LIN {X 0,Y 185.451,Z 180.384,A -85,B 0,C 180,E1 -22369.893,E2 -22369.893} C_VEL
LIN {X 0,Y 185.61,Z 180.474,A -85,B 0,C 180,E1 -22373.267,E2 -22373.267} C_VEL
LIN {X 0,Y 186.703,Z 185.931,A -85,B 0,C 180,E1 -22376.028,E2 -22376.028} C_VEL
LIN {X 0,Y 194.99,Z 213.07,A -85,B 0,C 180,E1 -22378.383,E2 -22378.383} C_VEL
LIN {X 0,Y 197.604,Z 239.191,A -85,B 0,C 180,E1 -22379.998,E2 -22379.998} C_VEL
LIN {X 0,Y 195.443,Z 280.522,A -85,B 0,C 180,E1 -22381.986,E2 -22381.986} C_VEL
LIN {X 0,Y 194.473,Z 286.295,A -85,B 0,C 180,E1 -22382.216,E2 -22382.216} C_VEL
LIN {X 0,Y 191.045,Z 295.55,A -85,B 0,C 180,E1 -22382.527,E2 -22382.527} C_VEL
LIN {X 0,Y 187.492,Z 304.682,A -85,B 0,C 180,E1 -22383.032,E2 -22383.032} C_VEL
LIN {X 0,Y 186.3,Z 310.262,A -85,B 0,C 180,E1 -22383.531,E2 -22383.531} C_VEL
LIN {X 0,Y 184.548,Z 324.129,A -85,B 0,C 180,E1 -22385.237,E2 -22385.237} C_VEL
LIN {X 0,Y 182.934,Z 335.61,A -85,B 0,C 180,E1 -22387.111,E2 -22387.111} C_VEL
LIN {X 0,Y 181.066,Z 347.271,A -85,B 0,C 180,E1 -22389.556,E2 -22389.556} C_VEL
LIN {X 0,Y 179.457,Z 357.77,A -85,B 0,C 180,E1 -22392.334,E2 -22392.334} C_VEL
LIN {X 0,Y 178.167,Z 366.277,A -85,B 0,C 180,E1 -22395.145,E2 -22395.145} C_VEL
LIN {X 0,Y 177.112,Z 374.602,A -85,B 0,C 180,E1 -22398.558,E2 -22398.558} C_VEL
LIN {X 0,Y 176.53,Z 381.268,A -85,B 0,C 180,E1 -22401.992,E2 -22401.992} C_VEL
LIN {X 0,Y 176.349,Z 386.5,A -85,B 0,C 180,E1 -22405.43,E2 -22405.43} C_VEL
LIN {X 0,Y 176.332,Z 390.477,A -85,B 0,C 180,E1 -22408.86,E2 -22408.86} C_VEL
LIN {X 0,Y 176.266,Z 393.307,A -85,B 0,C 180,E1 -22412.287,E2 -22412.287} C_VEL
LIN {X 0,Y 176.184,Z 395.515,A -85,B 0,C 180,E1 -22416.875,E2 -22416.875} C_VEL
LIN {X 0,Y 177.166,Z 396.208,A -85,B 0,C 180,E1 -22421.442,E2 -22421.442} C_VEL
LIN {X 0,Y 179.11,Z 395.354,A -85,B 0,C 180,E1 -22425.944,E2 -22425.944} C_VEL
LIN {X 0,Y 182.326,Z 392.981,A -85,B 0,C 180,E1 -22430.301,E2 -22430.301} C_VEL
LIN {X 0,Y 185.623,Z 390.146,A -85,B 0,C 180,E1 -22433.427,E2 -22433.427} C_VEL
LIN {X 0,Y 190.628,Z 384.946,A -85,B 0,C 180,E1 -22437.444,E2 -22437.444} C_VEL
LIN {X 0,Y 195.03,Z 379.819,A -85,B 0,C 180,E1 -22440.3,E2 -22440.3} C_VEL
LIN {X 0,Y 200.108,Z 373.441,A -85,B 0,C 180,E1 -22442.984,E2 -22442.984} C_VEL
LIN {X 0,Y 206.708,Z 364.199,A -85,B 0,C 180,E1 -22445.911,E2 -22445.911} C_VEL
LIN {X 0,Y 211.819,Z 356.151,A -85,B 0,C 180,E1 -22447.868,E2 -22447.868} C_VEL
LIN {X 0,Y 217.199,Z 346.506,A -85,B 0,C 180,E1 -22449.723,E2 -22449.723} C_VEL
LIN {X 0,Y 222.849,Z 334.573,A -85,B 0,C 180,E1 -22451.476,E2 -22451.476} C_VEL
LIN {X 0,Y 227.689,Z 322.728,A -85,B 0,C 180,E1 -22452.773,E2 -22452.773} C_VEL
LIN {X 0,Y 231.851,Z 310.219,A -85,B 0,C 180,E1 -22453.751,E2 -22453.751} C_VEL
LIN {X 0,Y 235.139,Z 297.091,A -85,B 0,C 180,E1 -22454.54,E2 -22454.54} C_VEL
LIN {X 0,Y 237.675,Z 281.593,A -85,B 0,C 180,E1 -22455.21,E2 -22455.21} C_VEL
LIN {X 0,Y 240.135,Z 263.541,A -85,B 0,C 180,E1 -22455.927,E2 -22455.927} C_VEL
LIN {X 0,Y 238.425,Z 258.199,A -85,B 0,C 180,E1 -22457.785,E2 -22457.785} C_VEL
LIN {X 0,Y 236.912,Z 254.032,A -85,B 0,C 180,E1 -22459.595,E2 -22459.595} C_VEL
LIN {X 0,Y 235.86,Z 251.223,A -85,B 0,C 180,E1 -22461.183,E2 -22461.183} C_VEL
LIN {X 0,Y 234.74,Z 248.234,A -85,B 0,C 180,E1 -22463.217,E2 -22463.217} C_VEL
LIN {X 0,Y 233.654,Z 245.558,A -85,B 0,C 180,E1 -22466.277,E2 -22466.277} C_VEL
LIN {X 0,Y 233.421,Z 244.65,A -85,B 0,C 180,E1 -22468.158,E2 -22468.158} C_VEL
LIN {X 0,Y 233.575,Z 244.599,A -85,B 0,C 180,E1 -22471.222,E2 -22471.222} C_VEL
LIN {X 0,Y 234.571,Z 246.09,A -85,B 0,C 180,E1 -22474.401,E2 -22474.401} C_VEL
LIN {X 0,Y 235.287,Z 247.149,A -85,B 0,C 180,E1 -22475.846,E2 -22475.846} C_VEL
LIN {X 0,Y 237.14,Z 250.744,A -85,B 0,C 180,E1 -22478.579,E2 -22478.579} C_VEL
LIN {X 0,Y 239.474,Z 255.65,A -85,B 0,C 180,E1 -22481.167,E2 -22481.167} C_VEL
LIN {X 0,Y 240.686,Z 258.623,A -85,B 0,C 180,E1 -22482.374,E2 -22482.374} C_VEL
LIN {X 0,Y 236.176,Z 289.327,A -85,B 0,C 180,E1 -22483.584,E2 -22483.584} C_VEL
LIN {X 0,Y 233.164,Z 302.706,A -85,B 0,C 180,E1 -22484.372,E2 -22484.372} C_VEL
LIN {X 0,Y 229.525,Z 314.723,A -85,B 0,C 180,E1 -22485.368,E2 -22485.368} C_VEL
LIN {X 0,Y 225.29,Z 326.032,A -85,B 0,C 180,E1 -22486.61,E2 -22486.61} C_VEL
LIN {X 0,Y 220.162,Z 337.516,A -85,B 0,C 180,E1 -22488.259,E2 -22488.259} C_VEL
LIN {X 0,Y 214.619,Z 347.927,A -85,B 0,C 180,E1 -22490.19,E2 -22490.19} C_VEL
LIN {X 0,Y 209.255,Z 356.656,A -85,B 0,C 180,E1 -22492.28,E2 -22492.28} C_VEL
LIN {X 0,Y 204.148,Z 363.965,A -85,B 0,C 180,E1 -22494.518,E2 -22494.518} C_VEL
LIN {X 0,Y 198.214,Z 371.419,A -85,B 0,C 180,E1 -22497.46,E2 -22497.46} C_VEL
LIN {X 0,Y 192.399,Z 377.919,A -85,B 0,C 180,E1 -22501.047,E2 -22501.047} C_VEL
LIN {X 0,Y 188.037,Z 382.07,A -85,B 0,C 180,E1 -22504.287,E2 -22504.287} C_VEL
LIN {X 0,Y 184.361,Z 385.041,A -85,B 0,C 180,E1 -22507.62,E2 -22507.62} C_VEL
LIN {X 0,Y 181.286,Z 386.968,A -85,B 0,C 180,E1 -22511.177,E2 -22511.177} C_VEL
LIN {X 0,Y 179.696,Z 387.622,A -85,B 0,C 180,E1 -22513.572,E2 -22513.572} C_VEL
LIN {X 0,Y 177.448,Z 387.679,A -85,B 0,C 180,E1 -22518.089,E2 -22518.089} C_VEL
LIN {X 0,Y 176.483,Z 386.859,A -85,B 0,C 180,E1 -22521.003,E2 -22521.003} C_VEL
LIN {X 0,Y 175.945,Z 385.646,A -85,B 0,C 180,E1 -22523.544,E2 -22523.544} C_VEL
LIN {X 0,Y 175.632,Z 383.889,A -85,B 0,C 180,E1 -22526.116,E2 -22526.116} C_VEL
LIN {X 0,Y 175.734,Z 380.218,A -85,B 0,C 180,E1 -22529.994,E2 -22529.994} C_VEL
LIN {X 0,Y 176.17,Z 375.043,A -85,B 0,C 180,E1 -22533.953,E2 -22533.953} C_VEL
LIN {X 0,Y 176.776,Z 369.274,A -85,B 0,C 180,E1 -22537.33,E2 -22537.33} C_VEL
LIN {X 0,Y 177.741,Z 361.636,A -85,B 0,C 180,E1 -22540.862,E2 -22540.862} C_VEL
LIN {X 0,Y 179.054,Z 352.651,A -85,B 0,C 180,E1 -22544.164,E2 -22544.164} C_VEL
LIN {X 0,Y 180.522,Z 343.259,A -85,B 0,C 180,E1 -22546.947,E2 -22546.947} C_VEL
LIN {X 0,Y 182.287,Z 331.812,A -85,B 0,C 180,E1 -22549.638,E2 -22549.638} C_VEL
LIN {X 0,Y 183.88,Z 321.431,A -85,B 0,C 180,E1 -22551.585,E2 -22551.585} C_VEL
LIN {X 0,Y 185.496,Z 309.195,A -85,B 0,C 180,E1 -22553.394,E2 -22553.394} C_VEL
LIN {X 0,Y 186.884,Z 295.677,A -85,B 0,C 180,E1 -22554.88,E2 -22554.88} C_VEL
LIN {X 0,Y 187.935,Z 282.298,A -85,B 0,C 180,E1 -22555.898,E2 -22555.898} C_VEL
LIN {X 0,Y 191.478,Z 219.149,A -85,B 0,C 180,E1 -22559.077,E2 -22559.077} C_VEL
LIN {X 0,Y 184.988,Z 198.355,A -85,B 0,C 180,E1 -22560.871,E2 -22560.871} C_VEL
LIN {X 0,Y 178.472,Z 181.316,A -85,B 0,C 180,E1 -22562.595,E2 -22562.595} C_VEL
LIN {X 0,Y 178.468,Z 181.254,A -85,B 0,C 180,E1 -22566.807,E2 -22566.807} C_VEL
LIN {X 0,Y 178.61,Z 181.237,A -85,B 0,C 180,E1 -22571.65,E2 -22571.65} C_VEL
LIN {X 0,Y 178.631,Z 181.236,A -85,B 0,C 180,E1 -22576.344,E2 -22576.344} C_VEL
LIN {X 0,Y 178.909,Z 181.198,A -85,B 0,C 180,E1 -22580.958,E2 -22580.958} C_VEL
LIN {X 0,Y 179.127,Z 181.172,A -85,B 0,C 180,E1 -22587.75,E2 -22587.75} C_VEL
LIN {X 0,Y 179.348,Z 181.141,A -85,B 0,C 180,E1 -22589.998,E2 -22589.998} C_VEL
LIN {X 0,Y 178.836,Z 181.207,A -85,B 0,C 180,E1 -22594.506,E2 -22594.506} C_VEL
LIN {X 0,Y 178.905,Z 181.194,A -85,B 0,C 180,E1 -22599.039,E2 -22599.039} C_VEL
LIN {X 0,Y 178.628,Z 181.234,A -85,B 0,C 180,E1 -22603.652,E2 -22603.652} C_VEL
LIN {X 0,Y 178.555,Z 181.242,A -85,B 0,C 180,E1 -22609.15,E2 -22609.15} C_VEL
LIN {X 0,Y 178.465,Z 181.251,A -85,B 0,C 180,E1 -22615.074,E2 -22615.074} C_VEL
LIN {X 0,Y 178.459,Z 181.255,A -85,B 0,C 180,E1 -22620.792,E2 -22620.792} C_VEL
LIN {X 0,Y 178.481,Z 181.247,A -85,B 0,C 180,E1 -22624.216,E2 -22624.216} C_VEL
LIN {X 0,Y 178.385,Z 181.265,A -85,B 0,C 180,E1 -22629.075,E2 -22629.075} C_VEL
LIN {X 0,Y 178.39,Z 181.257,A -85,B 0,C 180,E1 -22632.044,E2 -22632.044} C_VEL
LIN {X 0,Y 178.388,Z 181.265,A -85,B 0,C 180,E1 -22635.163,E2 -22635.163} C_VEL
LIN {X 0,Y 178.394,Z 181.263,A -85,B 0,C 180,E1 -22638.46,E2 -22638.46} C_VEL
LIN {X 0,Y 178.415,Z 181.259,A -85,B 0,C 180,E1 -22643.78,E2 -22643.78} C_VEL
LIN {X 0,Y 178.479,Z 181.253,A -85,B 0,C 180,E1 -22646.544,E2 -22646.544} C_VEL
LIN {X 0,Y 178.435,Z 181.257,A -85,B 0,C 180,E1 -22651.793,E2 -22651.793} C_VEL
LIN {X 0,Y 178.5,Z 181.248,A -85,B 0,C 180,E1 -22654.895,E2 -22654.895} C_VEL
LIN {X 0,Y 178.6,Z 181.237,A -85,B 0,C 180,E1 -22661.65,E2 -22661.65} C_VEL
LIN {X 0,Y 178.62,Z 181.233,A -85,B 0,C 180,E1 -22666.344,E2 -22666.344} C_VEL
LIN {X 0,Y 178.899,Z 181.199,A -85,B 0,C 180,E1 -22670.959,E2 -22670.959} C_VEL
LIN {X 0,Y 179.117,Z 181.174,A -85,B 0,C 180,E1 -22677.751,E2 -22677.751} C_VEL
LIN {X 0,Y 179.338,Z 181.145,A -85,B 0,C 180,E1 -22679.999,E2 -22679.999} C_VEL
LIN {X 0,Y 178.826,Z 181.208,A -85,B 0,C 180,E1 -22684.508,E2 -22684.508} C_VEL
LIN {X 0,Y 178.896,Z 181.198,A -85,B 0,C 180,E1 -22689.041,E2 -22689.041} C_VEL
LIN {X 0,Y 178.619,Z 181.236,A -85,B 0,C 180,E1 -22693.655,E2 -22693.655} C_VEL
LIN {X 0,Y 178.548,Z 181.24,A -85,B 0,C 180,E1 -22699.152,E2 -22699.152} C_VEL
LIN {X 0,Y 178.459,Z 181.255,A -85,B 0,C 180,E1 -22705.077,E2 -22705.077} C_VEL
LIN {X 0,Y 178.454,Z 181.255,A -85,B 0,C 180,E1 -22710.795,E2 -22710.795} C_VEL
LIN {X 0,Y 178.476,Z 181.25,A -85,B 0,C 180,E1 -22714.219,E2 -22714.219} C_VEL
LIN {X 0,Y 178.381,Z 181.265,A -85,B 0,C 180,E1 -22719.078,E2 -22719.078} C_VEL
LIN {X 0,Y 178.387,Z 181.261,A -85,B 0,C 180,E1 -22722.048,E2 -22722.048} C_VEL
LIN {X 0,Y 178.386,Z 181.267,A -85,B 0,C 180,E1 -22725.166,E2 -22725.166} C_VEL
LIN {X 0,Y 178.392,Z 181.264,A -85,B 0,C 180,E1 -22728.463,E2 -22728.463} C_VEL
LIN {X 0,Y 178.548,Z 181.257,A -85,B 0,C 180,E1 -22732.828,E2 -22732.828} C_VEL
LIN {X 0,Y 179.513,Z 185.981,A -85,B 0,C 180,E1 -22735.227,E2 -22735.227} C_VEL
LIN {X 0,Y 188.36,Z 214.966,A -85,B 0,C 180,E1 -22737.833,E2 -22737.833} C_VEL
LIN {X 0,Y 190.739,Z 240.435,A -85,B 0,C 180,E1 -22739.459,E2 -22739.459} C_VEL
LIN {X 0,Y 187.702,Z 294.949,A -85,B 0,C 180,E1 -22742.247,E2 -22742.247} C_VEL
LIN {X 0,Y 186.444,Z 309.054,A -85,B 0,C 180,E1 -22743.411,E2 -22743.411} C_VEL
LIN {X 0,Y 186.3,Z 310.262,A -85,B 0,C 180,E1 -22743.531,E2 -22743.531} C_VEL
LIN {X 0,Y 184.978,Z 315.739,A -85,B 0,C 180,E1 -22744.087,E2 -22744.087} C_VEL
LIN {X 0,Y 181.018,Z 324.289,A -85,B 0,C 180,E1 -22745.068,E2 -22745.068} C_VEL
LIN {X 0,Y 176.974,Z 332.538,A -85,B 0,C 180,E1 -22746.295,E2 -22746.295} C_VEL
LIN {X 0,Y 175.539,Z 337.528,A -85,B 0,C 180,E1 -22747.221,E2 -22747.221} C_VEL
LIN {X 0,Y 173.85,Z 348.124,A -85,B 0,C 180,E1 -22749.596,E2 -22749.596} C_VEL
LIN {X 0,Y 172.373,Z 357.468,A -85,B 0,C 180,E1 -22752.197,E2 -22752.197} C_VEL
LIN {X 0,Y 171.057,Z 365.993,A -85,B 0,C 180,E1 -22755.123,E2 -22755.123} C_VEL
LIN {X 0,Y 170.019,Z 374.338,A -85,B 0,C 180,E1 -22758.679,E2 -22758.679} C_VEL
LIN {X 0,Y 169.512,Z 379.97,A -85,B 0,C 180,E1 -22761.658,E2 -22761.658} C_VEL
LIN {X 0,Y 169.295,Z 385.409,A -85,B 0,C 180,E1 -22765.24,E2 -22765.24} C_VEL
LIN {X 0,Y 169.279,Z 389.572,A -85,B 0,C 180,E1 -22768.813,E2 -22768.813} C_VEL
LIN {X 0,Y 169.198,Z 392.583,A -85,B 0,C 180,E1 -22772.383,E2 -22772.383} C_VEL
LIN {X 0,Y 169.039,Z 394.032,A -85,B 0,C 180,E1 -22774.772,E2 -22774.772} C_VEL
LIN {X 0,Y 169.129,Z 395.073,A -85,B 0,C 180,E1 -22777.163,E2 -22777.163} C_VEL
LIN {X 0,Y 170.184,Z 395.952,A -85,B 0,C 180,E1 -22781.918,E2 -22781.918} C_VEL
LIN {X 0,Y 172.265,Z 395.359,A -85,B 0,C 180,E1 -22786.596,E2 -22786.596} C_VEL
LIN {X 0,Y 173.807,Z 394.504,A -85,B 0,C 180,E1 -22788.876,E2 -22788.876} C_VEL
LIN {X 0,Y 177.963,Z 391.591,A -85,B 0,C 180,E1 -22793.263,E2 -22793.263} C_VEL
LIN {X 0,Y 182.975,Z 387.134,A -85,B 0,C 180,E1 -22797.448,E2 -22797.448} C_VEL
LIN {X 0,Y 187.391,Z 382.606,A -85,B 0,C 180,E1 -22800.419,E2 -22800.419} C_VEL
LIN {X 0,Y 193.364,Z 375.929,A -85,B 0,C 180,E1 -22803.663,E2 -22803.663} C_VEL
LIN {X 0,Y 200.141,Z 367.459,A -85,B 0,C 180,E1 -22806.654,E2 -22806.654} C_VEL
LIN {X 0,Y 206.443,Z 358.412,A -85,B 0,C 180,E1 -22809.037,E2 -22809.037} C_VEL
LIN {X 0,Y 213.139,Z 347.295,A -85,B 0,C 180,E1 -22811.262,E2 -22811.262} C_VEL
LIN {X 0,Y 218.411,Z 337.106,A -85,B 0,C 180,E1 -22812.826,E2 -22812.826} C_VEL
LIN {X 0,Y 223.4,Z 325.833,A -85,B 0,C 180,E1 -22814.112,E2 -22814.112} C_VEL
LIN {X 0,Y 227.963,Z 313.355,A -85,B 0,C 180,E1 -22815.162,E2 -22815.162} C_VEL
LIN {X 0,Y 231.687,Z 299.909,A -85,B 0,C 180,E1 -22816.014,E2 -22816.014} C_VEL
LIN {X 0,Y 234.426,Z 286.088,A -85,B 0,C 180,E1 -22816.635,E2 -22816.635} C_VEL
LIN {X 0,Y 237.134,Z 267.255,A -85,B 0,C 180,E1 -22817.403,E2 -22817.403} C_VEL
LIN {X 0,Y 235.477,Z 261.867,A -85,B 0,C 180,E1 -22819.489,E2 -22819.489} C_VEL
LIN {X 0,Y 234.173,Z 257.979,A -85,B 0,C 180,E1 -22821.561,E2 -22821.561} C_VEL
LIN {X 0,Y 233.184,Z 255.014,A -85,B 0,C 180,E1 -22823.577,E2 -22823.577} C_VEL
LIN {X 0,Y 232.217,Z 252.288,A -85,B 0,C 180,E1 -22826.767,E2 -22826.767} C_VEL
LIN {X 0,Y 231.999,Z 251.475,A -85,B 0,C 180,E1 -22829.004,E2 -22829.004} C_VEL
LIN {X 0,Y 232.373,Z 251.836,A -85,B 0,C 180,E1 -22832.071,E2 -22832.071} C_VEL
LIN {X 0,Y 233.663,Z 253.817,A -85,B 0,C 180,E1 -22835.382,E2 -22835.382} C_VEL
LIN {X 0,Y 235.34,Z 257.377,A -85,B 0,C 180,E1 -22838.103,E2 -22838.103} C_VEL
LIN {X 0,Y 237.32,Z 261.821,A -85,B 0,C 180,E1 -22840.504,E2 -22840.504} C_VEL
LIN {X 0,Y 237.707,Z 262.858,A -85,B 0,C 180,E1 -22840.939,E2 -22840.939} C_VEL
LIN {X 0,Y 233.439,Z 289.877,A -85,B 0,C 180,E1 -22841.995,E2 -22841.995} C_VEL
LIN {X 0,Y 230.262,Z 303.162,A -85,B 0,C 180,E1 -22842.772,E2 -22842.772} C_VEL
LIN {X 0,Y 226.388,Z 315.434,A -85,B 0,C 180,E1 -22843.776,E2 -22843.776} C_VEL
LIN {X 0,Y 221.725,Z 327.318,A -85,B 0,C 180,E1 -22845.076,E2 -22845.076} C_VEL
LIN {X 0,Y 216.772,Z 337.743,A -85,B 0,C 180,E1 -22846.571,E2 -22846.571} C_VEL
LIN {X 0,Y 210.976,Z 348.019,A -85,B 0,C 180,E1 -22848.471,E2 -22848.471} C_VEL
LIN {X 0,Y 205.104,Z 357.104,A -85,B 0,C 180,E1 -22850.633,E2 -22850.633} C_VEL
LIN {X 0,Y 198.669,Z 365.689,A -85,B 0,C 180,E1 -22853.334,E2 -22853.334} C_VEL
LIN {X 0,Y 193.399,Z 371.78,A -85,B 0,C 180,E1 -22855.833,E2 -22855.833} C_VEL
LIN {X 0,Y 188.003,Z 377.408,A -85,B 0,C 180,E1 -22858.929,E2 -22858.929} C_VEL
LIN {X 0,Y 182.893,Z 382,A -85,B 0,C 180,E1 -22862.394,E2 -22862.394} C_VEL
LIN {X 0,Y 180.269,Z 384.023,A -85,B 0,C 180,E1 -22864.473,E2 -22864.473} C_VEL
LIN {X 0,Y 177.186,Z 386.081,A -85,B 0,C 180,E1 -22867.413,E2 -22867.413} C_VEL
LIN {X 0,Y 173.706,Z 387.76,A -85,B 0,C 180,E1 -22871.672,E2 -22871.672} C_VEL
LIN {X 0,Y 172.112,Z 388.066,A -85,B 0,C 180,E1 -22874.183,E2 -22874.183} C_VEL
LIN {X 0,Y 170.235,Z 387.622,A -85,B 0,C 180,E1 -22878.274,E2 -22878.274} C_VEL
LIN {X 0,Y 169.152,Z 386.232,A -85,B 0,C 180,E1 -22881.959,E2 -22881.959} C_VEL
LIN {X 0,Y 168.56,Z 383.621,A -85,B 0,C 180,E1 -22885.964,E2 -22885.964} C_VEL
LIN {X 0,Y 168.652,Z 379.764,A -85,B 0,C 180,E1 -22890.005,E2 -22890.005} C_VEL
LIN {X 0,Y 169.046,Z 374.941,A -85,B 0,C 180,E1 -22893.745,E2 -22893.745} C_VEL
LIN {X 0,Y 169.727,Z 368.633,A -85,B 0,C 180,E1 -22897.522,E2 -22897.522} C_VEL
LIN {X 0,Y 170.732,Z 360.824,A -85,B 0,C 180,E1 -22901.196,E2 -22901.196} C_VEL
LIN {X 0,Y 172.003,Z 352.301,A -85,B 0,C 180,E1 -22904.406,E2 -22904.406} C_VEL
LIN {X 0,Y 173.493,Z 342.963,A -85,B 0,C 180,E1 -22907.243,E2 -22907.243} C_VEL
LIN {X 0,Y 175.382,Z 331.03,A -85,B 0,C 180,E1 -22910.119,E2 -22910.119} C_VEL
LIN {X 0,Y 177.023,Z 320.439,A -85,B 0,C 180,E1 -22912.139,E2 -22912.139} C_VEL
LIN {X 0,Y 178.669,Z 307.992,A -85,B 0,C 180,E1 -22913.985,E2 -22913.985} C_VEL
LIN {X 0,Y 179.945,Z 295.833,A -85,B 0,C 180,E1 -22915.35,E2 -22915.35} C_VEL
LIN {X 0,Y 181.03,Z 282.582,A -85,B 0,C 180,E1 -22916.395,E2 -22916.395} C_VEL
LIN {X 0,Y 184.658,Z 220.397,A -85,B 0,C 180,E1 -22919.648,E2 -22919.648} C_VEL
LIN {X 0,Y 178.39,Z 200.423,A -85,B 0,C 180,E1 -22921.463,E2 -22921.463} C_VEL
LIN {X 0,Y 171.445,Z 182.365,A -85,B 0,C 180,E1 -22923.382,E2 -22923.382} C_VEL
LIN {X 0,Y 171.394,Z 182.136,A -85,B 0,C 180,E1 -22923.559,E2 -22923.559} C_VEL
LIN {X 0,Y 171.42,Z 182.134,A -85,B 0,C 180,E1 -22928.345,E2 -22928.345} C_VEL
LIN {X 0,Y 171.513,Z 182.121,A -85,B 0,C 180,E1 -22930.862,E2 -22930.862} C_VEL
LIN {X 0,Y 171.546,Z 182.117,A -85,B 0,C 180,E1 -22935.768,E2 -22935.768} C_VEL
LIN {X 0,Y 171.848,Z 182.078,A -85,B 0,C 180,E1 -22940.583,E2 -22940.583} C_VEL
LIN {X 0,Y 171.787,Z 182.085,A -85,B 0,C 180,E1 -22945.305,E2 -22945.305} C_VEL
LIN {X 0,Y 172.313,Z 182.017,A -85,B 0,C 180,E1 -22949.998,E2 -22949.998} C_VEL
LIN {X 0,Y 171.785,Z 182.085,A -85,B 0,C 180,E1 -22954.691,E2 -22954.691} C_VEL
LIN {X 0,Y 171.844,Z 182.075,A -85,B 0,C 180,E1 -22959.413,E2 -22959.413} C_VEL
LIN {X 0,Y 171.543,Z 182.115,A -85,B 0,C 180,E1 -22964.228,E2 -22964.228} C_VEL
LIN {X 0,Y 171.48,Z 182.125,A -85,B 0,C 180,E1 -22969.497,E2 -22969.497} C_VEL
LIN {X 0,Y 171.403,Z 182.131,A -85,B 0,C 180,E1 -22975.567,E2 -22975.567} C_VEL
LIN {X 0,Y 171.416,Z 182.132,A -85,B 0,C 180,E1 -22980.57,E2 -22980.57} C_VEL
LIN {X 0,Y 171.39,Z 182.133,A -85,B 0,C 180,E1 -22985.033,E2 -22985.033} C_VEL
LIN {X 0,Y 171.341,Z 182.143,A -85,B 0,C 180,E1 -22988.799,E2 -22988.799} C_VEL
LIN {X 0,Y 171.315,Z 182.143,A -85,B 0,C 180,E1 -22994.216,E2 -22994.216} C_VEL
LIN {X 0,Y 171.326,Z 182.141,A -85,B 0,C 180,E1 -22998.978,E2 -22998.978} C_VEL
LIN {X 0,Y 171.356,Z 182.137,A -85,B 0,C 180,E1 -23002.032,E2 -23002.032} C_VEL
LIN {X 0,Y 171.393,Z 182.135,A -85,B 0,C 180,E1 -23005.091,E2 -23005.091} C_VEL
LIN {X 0,Y 171.403,Z 182.133,A -85,B 0,C 180,E1 -23010.525,E2 -23010.525} C_VEL
LIN {X 0,Y 171.421,Z 182.129,A -85,B 0,C 180,E1 -23015.795,E2 -23015.795} C_VEL
LIN {X 0,Y 171.501,Z 182.122,A -85,B 0,C 180,E1 -23020.862,E2 -23020.862} C_VEL
LIN {X 0,Y 171.536,Z 182.112,A -85,B 0,C 180,E1 -23025.769,E2 -23025.769} C_VEL
LIN {X 0,Y 171.837,Z 182.079,A -85,B 0,C 180,E1 -23030.584,E2 -23030.584} C_VEL
LIN {X 0,Y 171.777,Z 182.084,A -85,B 0,C 180,E1 -23035.306,E2 -23035.306} C_VEL
LIN {X 0,Y 172.303,Z 182.021,A -85,B 0,C 180,E1 -23039.999,E2 -23039.999} C_VEL
LIN {X 0,Y 171.775,Z 182.086,A -85,B 0,C 180,E1 -23044.693,E2 -23044.693} C_VEL
LIN {X 0,Y 171.835,Z 182.079,A -85,B 0,C 180,E1 -23049.415,E2 -23049.415} C_VEL
LIN {X 0,Y 171.535,Z 182.117,A -85,B 0,C 180,E1 -23054.23,E2 -23054.23} C_VEL
LIN {X 0,Y 171.472,Z 182.122,A -85,B 0,C 180,E1 -23059.499,E2 -23059.499} C_VEL
LIN {X 0,Y 171.396,Z 182.133,A -85,B 0,C 180,E1 -23065.57,E2 -23065.57} C_VEL
LIN {X 0,Y 171.411,Z 182.132,A -85,B 0,C 180,E1 -23070.573,E2 -23070.573} C_VEL
LIN {X 0,Y 171.386,Z 182.133,A -85,B 0,C 180,E1 -23075.036,E2 -23075.036} C_VEL
LIN {X 0,Y 171.337,Z 182.141,A -85,B 0,C 180,E1 -23078.802,E2 -23078.802} C_VEL
LIN {X 0,Y 171.313,Z 182.145,A -85,B 0,C 180,E1 -23084.22,E2 -23084.22} C_VEL
LIN {X 0,Y 171.331,Z 182.145,A -85,B 0,C 180,E1 -23088.983,E2 -23088.983} C_VEL
LIN {X 0,Y 171.508,Z 182.251,A -85,B 0,C 180,E1 -23092.497,E2 -23092.497} C_VEL
LIN {X 0,Y 172.164,Z 185.558,A -85,B 0,C 180,E1 -23094.317,E2 -23094.317} C_VEL
LIN {X 0,Y 181.585,Z 216.234,A -85,B 0,C 180,E1 -23097.236,E2 -23097.236} C_VEL
LIN {X 0,Y 183.928,Z 240.636,A -85,B 0,C 180,E1 -23098.865,E2 -23098.865} C_VEL
LIN {X 0,Y 180.825,Z 294.391,A -85,B 0,C 180,E1 -23101.729,E2 -23101.729} C_VEL
LIN {X 0,Y 179.534,Z 308.569,A -85,B 0,C 180,E1 -23102.933,E2 -23102.933} C_VEL
LIN {X 0,Y 177.851,Z 321.835,A -85,B 0,C 180,E1 -23104.551,E2 -23104.551} C_VEL
LIN {X 0,Y 176.19,Z 333.749,A -85,B 0,C 180,E1 -23106.494,E2 -23106.494} C_VEL
LIN {X 0,Y 175.539,Z 337.528,A -85,B 0,C 180,E1 -23107.221,E2 -23107.221} C_VEL
LIN {X 0,Y 174.103,Z 342.397,A -85,B 0,C 180,E1 -23108.217,E2 -23108.217} C_VEL
LIN {X 0,Y 170.033,Z 349.848,A -85,B 0,C 180,E1 -23109.934,E2 -23109.934} C_VEL
LIN {X 0,Y 166.024,Z 356.816,A -85,B 0,C 180,E1 -23111.934,E2 -23111.934} C_VEL
LIN {X 0,Y 164.712,Z 360.93,A -85,B 0,C 180,E1 -23113.341,E2 -23113.341} C_VEL
LIN {X 0,Y 163.358,Z 370.011,A -85,B 0,C 180,E1 -23116.948,E2 -23116.948} C_VEL
LIN {X 0,Y 162.615,Z 377.488,A -85,B 0,C 180,E1 -23120.675,E2 -23120.675} C_VEL
LIN {X 0,Y 162.298,Z 382.505,A -85,B 0,C 180,E1 -23123.787,E2 -23123.787} C_VEL
LIN {X 0,Y 162.244,Z 387.316,A -85,B 0,C 180,E1 -23127.519,E2 -23127.519} C_VEL
LIN {X 0,Y 162.24,Z 389.86,A -85,B 0,C 180,E1 -23130.002,E2 -23130.002} C_VEL
LIN {X 0,Y 161.983,Z 392.671,A -85,B 0,C 180,E1 -23133.71,E2 -23133.71} C_VEL
LIN {X 0,Y 162.098,Z 394.534,A -85,B 0,C 180,E1 -23137.476,E2 -23137.476} C_VEL
LIN {X 0,Y 163.225,Z 395.693,A -85,B 0,C 180,E1 -23142.434,E2 -23142.434} C_VEL
LIN {X 0,Y 165.447,Z 395.307,A -85,B 0,C 180,E1 -23147.301,E2 -23147.301} C_VEL
LIN {X 0,Y 169.103,Z 393.479,A -85,B 0,C 180,E1 -23151.967,E2 -23151.967} C_VEL
LIN {X 0,Y 171.491,Z 391.995,A -85,B 0,C 180,E1 -23154.196,E2 -23154.196} C_VEL
LIN {X 0,Y 176.728,Z 387.778,A -85,B 0,C 180,E1 -23158.505,E2 -23158.505} C_VEL
LIN {X 0,Y 181.368,Z 383.558,A -85,B 0,C 180,E1 -23161.543,E2 -23161.543} C_VEL
LIN {X 0,Y 187.591,Z 377.251,A -85,B 0,C 180,E1 -23164.845,E2 -23164.845} C_VEL
LIN {X 0,Y 193.59,Z 370.456,A -85,B 0,C 180,E1 -23167.453,E2 -23167.453} C_VEL
LIN {X 0,Y 200.024,Z 362.238,A -85,B 0,C 180,E1 -23169.886,E2 -23169.886} C_VEL
LIN {X 0,Y 206.894,Z 352.111,A -85,B 0,C 180,E1 -23172.138,E2 -23172.138} C_VEL
LIN {X 0,Y 212.875,Z 341.811,A -85,B 0,C 180,E1 -23173.894,E2 -23173.894} C_VEL
LIN {X 0,Y 218.568,Z 330.325,A -85,B 0,C 180,E1 -23175.353,E2 -23175.353} C_VEL
LIN {X 0,Y 223.207,Z 319.278,A -85,B 0,C 180,E1 -23176.403,E2 -23176.403} C_VEL
LIN {X 0,Y 227.608,Z 306.194,A -85,B 0,C 180,E1 -23177.332,E2 -23177.332} C_VEL
LIN {X 0,Y 231.046,Z 292.161,A -85,B 0,C 180,E1 -23178.041,E2 -23178.041} C_VEL
LIN {X 0,Y 234.386,Z 271.211,A -85,B 0,C 180,E1 -23178.864,E2 -23178.864} C_VEL
LIN {X 0,Y 233.018,Z 266.387,A -85,B 0,C 180,E1 -23181.018,E2 -23181.018} C_VEL
LIN {X 0,Y 231.649,Z 261.786,A -85,B 0,C 180,E1 -23183.924,E2 -23183.924} C_VEL
LIN {X 0,Y 230.821,Z 259.194,A -85,B 0,C 180,E1 -23186.995,E2 -23186.995} C_VEL
LIN {X 0,Y 230.659,Z 258.477,A -85,B 0,C 180,E1 -23188.804,E2 -23188.804} C_VEL
LIN {X 0,Y 230.988,Z 258.777,A -85,B 0,C 180,E1 -23191.93,E2 -23191.93} C_VEL
LIN {X 0,Y 232.152,Z 260.749,A -85,B 0,C 180,E1 -23195.14,E2 -23195.14} C_VEL
LIN {X 0,Y 233.627,Z 264.097,A -85,B 0,C 180,E1 -23197.711,E2 -23197.711} C_VEL
LIN {X 0,Y 234.856,Z 267.276,A -85,B 0,C 180,E1 -23199.458,E2 -23199.458} C_VEL
LIN {X 0,Y 231.009,Z 290.555,A -85,B 0,C 180,E1 -23200.357,E2 -23200.357} C_VEL
LIN {X 0,Y 227.791,Z 303.503,A -85,B 0,C 180,E1 -23201.098,E2 -23201.098} C_VEL
LIN {X 0,Y 223.556,Z 316.172,A -85,B 0,C 180,E1 -23202.122,E2 -23202.122} C_VEL
LIN {X 0,Y 218.614,Z 328.041,A -85,B 0,C 180,E1 -23203.423,E2 -23203.423} C_VEL
LIN {X 0,Y 213.191,Z 338.777,A -85,B 0,C 180,E1 -23204.956,E2 -23204.956} C_VEL
LIN {X 0,Y 207.341,Z 348.666,A -85,B 0,C 180,E1 -23206.774,E2 -23206.774} C_VEL
LIN {X 0,Y 201.095,Z 357.757,A -85,B 0,C 180,E1 -23208.955,E2 -23208.955} C_VEL
LIN {X 0,Y 194.206,Z 366.295,A -85,B 0,C 180,E1 -23211.677,E2 -23211.677} C_VEL
LIN {X 0,Y 187.74,Z 373.271,A -85,B 0,C 180,E1 -23214.63,E2 -23214.63} C_VEL
LIN {X 0,Y 182.081,Z 378.629,A -85,B 0,C 180,E1 -23217.788,E2 -23217.788} C_VEL
LIN {X 0,Y 177.166,Z 382.574,A -85,B 0,C 180,E1 -23220.999,E2 -23220.999} C_VEL
LIN {X 0,Y 172.579,Z 385.649,A -85,B 0,C 180,E1 -23224.672,E2 -23224.672} C_VEL
LIN {X 0,Y 170.012,Z 387.004,A -85,B 0,C 180,E1 -23227.185,E2 -23227.185} C_VEL
LIN {X 0,Y 167.902,Z 387.863,A -85,B 0,C 180,E1 -23229.639,E2 -23229.639} C_VEL
LIN {X 0,Y 165.743,Z 388.299,A -85,B 0,C 180,E1 -23232.761,E2 -23232.761} C_VEL
LIN {X 0,Y 163.354,Z 387.746,A -85,B 0,C 180,E1 -23237.528,E2 -23237.528} C_VEL
LIN {X 0,Y 162.446,Z 386.779,A -85,B 0,C 180,E1 -23240.25,E2 -23240.25} C_VEL
LIN {X 0,Y 161.665,Z 384.617,A -85,B 0,C 180,E1 -23244.083,E2 -23244.083} C_VEL
LIN {X 0,Y 161.505,Z 380.779,A -85,B 0,C 180,E1 -23248.6,E2 -23248.6} C_VEL
LIN {X 0,Y 161.849,Z 375.697,A -85,B 0,C 180,E1 -23252.875,E2 -23252.875} C_VEL
LIN {X 0,Y 162.44,Z 370.09,A -85,B 0,C 180,E1 -23256.51,E2 -23256.51} C_VEL
LIN {X 0,Y 163.321,Z 362.959,A -85,B 0,C 180,E1 -23260.203,E2 -23260.203} C_VEL
LIN {X 0,Y 164.667,Z 353.792,A -85,B 0,C 180,E1 -23263.948,E2 -23263.948} C_VEL
LIN {X 0,Y 166.096,Z 345.142,A -85,B 0,C 180,E1 -23266.803,E2 -23266.803} C_VEL
LIN {X 0,Y 167.894,Z 333.796,A -85,B 0,C 180,E1 -23269.814,E2 -23269.814} C_VEL
LIN {X 0,Y 169.833,Z 321.676,A -85,B 0,C 180,E1 -23272.32,E2 -23272.32} C_VEL
LIN {X 0,Y 171.547,Z 309.484,A -85,B 0,C 180,E1 -23274.262,E2 -23274.262} C_VEL
LIN {X 0,Y 172.949,Z 296.709,A -85,B 0,C 180,E1 -23275.783,E2 -23275.783} C_VEL
LIN {X 0,Y 174.033,Z 283.689,A -85,B 0,C 180,E1 -23276.885,E2 -23276.885} C_VEL
LIN {X 0,Y 177.806,Z 221.62,A -85,B 0,C 180,E1 -23280.267,E2 -23280.267} C_VEL
LIN {X 0,Y 171.897,Z 202.689,A -85,B 0,C 180,E1 -23282.069,E2 -23282.069} C_VEL
LIN {X 0,Y 164.414,Z 183.222,A -85,B 0,C 180,E1 -23284.216,E2 -23284.216} C_VEL
LIN {X 0,Y 164.361,Z 183.013,A -85,B 0,C 180,E1 -23284.683,E2 -23284.683} C_VEL
LIN {X 0,Y 164.421,Z 183.006,A -85,B 0,C 180,E1 -23290.116,E2 -23290.116} C_VEL
LIN {X 0,Y 164.476,Z 182.997,A -85,B 0,C 180,E1 -23295.143,E2 -23295.143} C_VEL
LIN {X 0,Y 164.769,Z 182.961,A -85,B 0,C 180,E1 -23300.174,E2 -23300.174} C_VEL
LIN {X 0,Y 164.824,Z 182.953,A -85,B 0,C 180,E1 -23302.649,E2 -23302.649} C_VEL
LIN {X 0,Y 165.277,Z 182.893,A -85,B 0,C 180,E1 -23309.998,E2 -23309.998} C_VEL
LIN {X 0,Y 164.821,Z 182.952,A -85,B 0,C 180,E1 -23317.347,E2 -23317.347} C_VEL
LIN {X 0,Y 164.703,Z 182.967,A -85,B 0,C 180,E1 -23321.055,E2 -23321.055} C_VEL
LIN {X 0,Y 164.429,Z 182.999,A -85,B 0,C 180,E1 -23327.407,E2 -23327.407} C_VEL
LIN {X 0,Y 164.42,Z 183.003,A -85,B 0,C 180,E1 -23329.994,E2 -23329.994} C_VEL
LIN {X 0,Y 164.338,Z 183.01,A -85,B 0,C 180,E1 -23336.092,E2 -23336.092} C_VEL
LIN {X 0,Y 164.352,Z 183.012,A -85,B 0,C 180,E1 -23341.212,E2 -23341.212} C_VEL
LIN {X 0,Y 164.278,Z 183.021,A -85,B 0,C 180,E1 -23346.791,E2 -23346.791} C_VEL
LIN {X 0,Y 164.283,Z 183.018,A -85,B 0,C 180,E1 -23349.916,E2 -23349.916} C_VEL
LIN {X 0,Y 164.277,Z 183.02,A -85,B 0,C 180,E1 -23353.34,E2 -23353.34} C_VEL
LIN {X 0,Y 164.257,Z 183.026,A -85,B 0,C 180,E1 -23356.796,E2 -23356.796} C_VEL
LIN {X 0,Y 164.285,Z 183.016,A -85,B 0,C 180,E1 -23360.353,E2 -23360.353} C_VEL
LIN {X 0,Y 164.321,Z 183.016,A -85,B 0,C 180,E1 -23364.349,E2 -23364.349} C_VEL
LIN {X 0,Y 164.362,Z 183.007,A -85,B 0,C 180,E1 -23369.128,E2 -23369.128} C_VEL
LIN {X 0,Y 164.381,Z 183.008,A -85,B 0,C 180,E1 -23374.687,E2 -23374.687} C_VEL
LIN {X 0,Y 164.411,Z 183.005,A -85,B 0,C 180,E1 -23380.116,E2 -23380.116} C_VEL
LIN {X 0,Y 164.465,Z 182.992,A -85,B 0,C 180,E1 -23385.143,E2 -23385.143} C_VEL
LIN {X 0,Y 164.759,Z 182.963,A -85,B 0,C 180,E1 -23390.175,E2 -23390.175} C_VEL
LIN {X 0,Y 164.814,Z 182.951,A -85,B 0,C 180,E1 -23392.65,E2 -23392.65} C_VEL
LIN {X 0,Y 165.267,Z 182.897,A -85,B 0,C 180,E1 -23399.999,E2 -23399.999} C_VEL
LIN {X 0,Y 164.811,Z 182.955,A -85,B 0,C 180,E1 -23407.349,E2 -23407.349} C_VEL
LIN {X 0,Y 164.694,Z 182.964,A -85,B 0,C 180,E1 -23411.057,E2 -23411.057} C_VEL
LIN {X 0,Y 164.421,Z 183.002,A -85,B 0,C 180,E1 -23417.409,E2 -23417.409} C_VEL
LIN {X 0,Y 164.412,Z 183.002,A -85,B 0,C 180,E1 -23419.996,E2 -23419.996} C_VEL
LIN {X 0,Y 164.332,Z 183.011,A -85,B 0,C 180,E1 -23426.095,E2 -23426.095} C_VEL
LIN {X 0,Y 164.351,Z 183.014,A -85,B 0,C 180,E1 -23431.218,E2 -23431.218} C_VEL
LIN {X 0,Y 164.274,Z 183.016,A -85,B 0,C 180,E1 -23436.794,E2 -23436.794} C_VEL
LIN {X 0,Y 164.28,Z 183.021,A -85,B 0,C 180,E1 -23439.919,E2 -23439.919} C_VEL
LIN {X 0,Y 164.274,Z 183.022,A -85,B 0,C 180,E1 -23443.343,E2 -23443.343} C_VEL
LIN {X 0,Y 164.255,Z 183.026,A -85,B 0,C 180,E1 -23446.799,E2 -23446.799} C_VEL
LIN {X 0,Y 164.409,Z 183.118,A -85,B 0,C 180,E1 -23452.088,E2 -23452.088} C_VEL
LIN {X 0,Y 164.897,Z 185.339,A -85,B 0,C 180,E1 -23453.37,E2 -23453.37} C_VEL
LIN {X 0,Y 172.786,Z 210.72,A -85,B 0,C 180,E1 -23455.957,E2 -23455.957} C_VEL
LIN {X 0,Y 175.078,Z 218.871,A -85,B 0,C 180,E1 -23456.712,E2 -23456.712} C_VEL
LIN {X 0,Y 177.083,Z 241.327,A -85,B 0,C 180,E1 -23458.263,E2 -23458.263} C_VEL
LIN {X 0,Y 173.898,Z 294.773,A -85,B 0,C 180,E1 -23461.24,E2 -23461.24} C_VEL
LIN {X 0,Y 172.642,Z 308.09,A -85,B 0,C 180,E1 -23462.418,E2 -23462.418} C_VEL
LIN {X 0,Y 170.905,Z 321.426,A -85,B 0,C 180,E1 -23464.095,E2 -23464.095} C_VEL
LIN {X 0,Y 169.216,Z 333.343,A -85,B 0,C 180,E1 -23466.106,E2 -23466.106} C_VEL
LIN {X 0,Y 167.42,Z 344.27,A -85,B 0,C 180,E1 -23468.452,E2 -23468.452} C_VEL
LIN {X 0,Y 165.64,Z 355.164,A -85,B 0,C 180,E1 -23471.447,E2 -23471.447} C_VEL
LIN {X 0,Y 164.712,Z 360.93,A -85,B 0,C 180,E1 -23473.341,E2 -23473.341} C_VEL
LIN {X 0,Y 163.455,Z 364.908,A -85,B 0,C 180,E1 -23474.823,E2 -23474.823} C_VEL
LIN {X 0,Y 159.752,Z 370.665,A -85,B 0,C 180,E1 -23477.357,E2 -23477.357} C_VEL
LIN {X 0,Y 156.267,Z 375.908,A -85,B 0,C 180,E1 -23480.16,E2 -23480.16} C_VEL
LIN {X 0,Y 155.383,Z 378.936,A -85,B 0,C 180,E1 -23482.011,E2 -23482.011} C_VEL
LIN {X 0,Y 155.199,Z 385.152,A -85,B 0,C 180,E1 -23486.444,E2 -23486.444} C_VEL
LIN {X 0,Y 155.193,Z 388.906,A -85,B 0,C 180,E1 -23490.002,E2 -23490.002} C_VEL
LIN {X 0,Y 154.952,Z 391.83,A -85,B 0,C 180,E1 -23493.778,E2 -23493.778} C_VEL
LIN {X 0,Y 155.083,Z 393.967,A -85,B 0,C 180,E1 -23497.816,E2 -23497.816} C_VEL
LIN {X 0,Y 156.288,Z 395.35,A -85,B 0,C 180,E1 -23502.996,E2 -23502.996} C_VEL
LIN {X 0,Y 158.659,Z 395.263,A -85,B 0,C 180,E1 -23508.066,E2 -23508.066} C_VEL
LIN {X 0,Y 162.557,Z 393.665,A -85,B 0,C 180,E1 -23512.901,E2 -23512.901} C_VEL
LIN {X 0,Y 167.668,Z 390.59,A -85,B 0,C 180,E1 -23517.459,E2 -23517.459} C_VEL
LIN {X 0,Y 172.861,Z 386.67,A -85,B 0,C 180,E1 -23521.171,E2 -23521.171} C_VEL
LIN {X 0,Y 179.016,Z 381.269,A -85,B 0,C 180,E1 -23524.701,E2 -23524.701} C_VEL
LIN {X 0,Y 186.001,Z 374.411,A -85,B 0,C 180,E1 -23527.881,E2 -23527.881} C_VEL
LIN {X 0,Y 192.518,Z 367.123,A -85,B 0,C 180,E1 -23530.391,E2 -23530.391} C_VEL
LIN {X 0,Y 199.448,Z 358.216,A -85,B 0,C 180,E1 -23532.714,E2 -23532.714} C_VEL
LIN {X 0,Y 206.804,Z 347.243,A -85,B 0,C 180,E1 -23534.845,E2 -23534.845} C_VEL
LIN {X 0,Y 212.528,Z 337.237,A -85,B 0,C 180,E1 -23536.336,E2 -23536.336} C_VEL
LIN {X 0,Y 217.9,Z 326.23,A -85,B 0,C 180,E1 -23537.546,E2 -23537.546} C_VEL
LIN {X 0,Y 223.06,Z 313.286,A -85,B 0,C 180,E1 -23538.574,E2 -23538.574} C_VEL
LIN {X 0,Y 226.639,Z 301.74,A -85,B 0,C 180,E1 -23539.299,E2 -23539.299} C_VEL
LIN {X 0,Y 229.842,Z 287.641,A -85,B 0,C 180,E1 -23539.927,E2 -23539.927} C_VEL
LIN {X 0,Y 231.807,Z 275.295,A -85,B 0,C 180,E1 -23540.455,E2 -23540.455} C_VEL
LIN {X 0,Y 230.714,Z 271.173,A -85,B 0,C 180,E1 -23542.549,E2 -23542.549} C_VEL
LIN {X 0,Y 230.028,Z 268.366,A -85,B 0,C 180,E1 -23544.514,E2 -23544.514} C_VEL
LIN {X 0,Y 229.438,Z 266.144,A -85,B 0,C 180,E1 -23547.144,E2 -23547.144} C_VEL
LIN {X 0,Y 229.278,Z 265.441,A -85,B 0,C 180,E1 -23549.126,E2 -23549.126} C_VEL
LIN {X 0,Y 229.658,Z 265.837,A -85,B 0,C 180,E1 -23552.092,E2 -23552.092} C_VEL
LIN {X 0,Y 230.652,Z 267.656,A -85,B 0,C 180,E1 -23554.896,E2 -23554.896} C_VEL
LIN {X 0,Y 231.946,Z 270.918,A -85,B 0,C 180,E1 -23557.364,E2 -23557.364} C_VEL
LIN {X 0,Y 232.276,Z 272.102,A -85,B 0,C 180,E1 -23557.952,E2 -23557.952} C_VEL
LIN {X 0,Y 228.916,Z 290.993,A -85,B 0,C 180,E1 -23558.671,E2 -23558.671} C_VEL
LIN {X 0,Y 225.439,Z 304.176,A -85,B 0,C 180,E1 -23559.413,E2 -23559.413} C_VEL
LIN {X 0,Y 220.777,Z 317.471,A -85,B 0,C 180,E1 -23560.474,E2 -23560.474} C_VEL
LIN {X 0,Y 215.406,Z 329.628,A -85,B 0,C 180,E1 -23561.808,E2 -23561.808} C_VEL
LIN {X 0,Y 210.061,Z 339.591,A -85,B 0,C 180,E1 -23563.228,E2 -23563.228} C_VEL
LIN {X 0,Y 203.63,Z 349.764,A -85,B 0,C 180,E1 -23565.107,E2 -23565.107} C_VEL
LIN {X 0,Y 197.47,Z 358.237,A -85,B 0,C 180,E1 -23567.148,E2 -23567.148} C_VEL
LIN {X 0,Y 191.277,Z 365.585,A -85,B 0,C 180,E1 -23569.414,E2 -23569.414} C_VEL
LIN {X 0,Y 184.383,Z 372.657,A -85,B 0,C 180,E1 -23572.331,E2 -23572.331} C_VEL
LIN {X 0,Y 178.098,Z 378.252,A -85,B 0,C 180,E1 -23575.474,E2 -23575.474} C_VEL
LIN {X 0,Y 172.53,Z 382.512,A -85,B 0,C 180,E1 -23578.833,E2 -23578.833} C_VEL
LIN {X 0,Y 167.689,Z 385.564,A -85,B 0,C 180,E1 -23582.403,E2 -23582.403} C_VEL
LIN {X 0,Y 162.844,Z 387.796,A -85,B 0,C 180,E1 -23586.944,E2 -23586.944} C_VEL
LIN {X 0,Y 160.224,Z 388.478,A -85,B 0,C 180,E1 -23590.106,E2 -23590.106} C_VEL
LIN {X 0,Y 158.475,Z 388.532,A -85,B 0,C 180,E1 -23592.812,E2 -23592.812} C_VEL
LIN {X 0,Y 156.997,Z 388.121,A -85,B 0,C 180,E1 -23595.581,E2 -23595.581} C_VEL
LIN {X 0,Y 155.808,Z 387.174,A -85,B 0,C 180,E1 -23598.688,E2 -23598.688} C_VEL
LIN {X 0,Y 155.064,Z 385.93,A -85,B 0,C 180,E1 -23601.26,E2 -23601.26} C_VEL
LIN {X 0,Y 154.427,Z 382.875,A -85,B 0,C 180,E1 -23605.692,E2 -23605.692} C_VEL
LIN {X 0,Y 154.519,Z 378.473,A -85,B 0,C 180,E1 -23610.207,E2 -23610.207} C_VEL
LIN {X 0,Y 154.967,Z 373.324,A -85,B 0,C 180,E1 -23614.194,E2 -23614.194} C_VEL
LIN {X 0,Y 155.763,Z 366.452,A -85,B 0,C 180,E1 -23618.346,E2 -23618.346} C_VEL
LIN {X 0,Y 156.867,Z 358.238,A -85,B 0,C 180,E1 -23622.225,E2 -23622.225} C_VEL
LIN {X 0,Y 158.36,Z 349.078,A -85,B 0,C 180,E1 -23625.696,E2 -23625.696} C_VEL
LIN {X 0,Y 159.978,Z 338.951,A -85,B 0,C 180,E1 -23628.776,E2 -23628.776} C_VEL
LIN {X 0,Y 161.829,Z 328.003,A -85,B 0,C 180,E1 -23631.419,E2 -23631.419} C_VEL
LIN {X 0,Y 163.708,Z 315.878,A -85,B 0,C 180,E1 -23633.729,E2 -23633.729} C_VEL
LIN {X 0,Y 165.266,Z 303.78,A -85,B 0,C 180,E1 -23635.482,E2 -23635.482} C_VEL
LIN {X 0,Y 166.606,Z 290.115,A -85,B 0,C 180,E1 -23636.94,E2 -23636.94} C_VEL
LIN {X 0,Y 167.801,Z 274.34,A -85,B 0,C 180,E1 -23638.01,E2 -23638.01} C_VEL
LIN {X 0,Y 171.028,Z 222.89,A -85,B 0,C 180,E1 -23640.916,E2 -23640.916} C_VEL
LIN {X 0,Y 165.429,Z 205.067,A -85,B 0,C 180,E1 -23642.67,E2 -23642.67} C_VEL
LIN {X 0,Y 157.3,Z 183.917,A -85,B 0,C 180,E1 -23645.147,E2 -23645.147} C_VEL
LIN {X 0,Y 157.365,Z 183.883,A -85,B 0,C 180,E1 -23649.7,E2 -23649.7} C_VEL
LIN {X 0,Y 157.41,Z 183.878,A -85,B 0,C 180,E1 -23654.459,E2 -23654.459} C_VEL
LIN {X 0,Y 157.691,Z 183.844,A -85,B 0,C 180,E1 -23659.729,E2 -23659.729} C_VEL
LIN {X 0,Y 157.763,Z 183.834,A -85,B 0,C 180,E1 -23662.318,E2 -23662.318} C_VEL
LIN {X 0,Y 158.239,Z 183.769,A -85,B 0,C 180,E1 -23669.998,E2 -23669.998} C_VEL
LIN {X 0,Y 157.759,Z 183.829,A -85,B 0,C 180,E1 -23677.678,E2 -23677.678} C_VEL
LIN {X 0,Y 157.632,Z 183.848,A -85,B 0,C 180,E1 -23681.221,E2 -23681.221} C_VEL
LIN {X 0,Y 157.407,Z 183.874,A -85,B 0,C 180,E1 -23685.537,E2 -23685.537} C_VEL
LIN {X 0,Y 157.304,Z 183.89,A -85,B 0,C 180,E1 -23690.94,E2 -23690.94} C_VEL
LIN {X 0,Y 157.266,Z 183.891,A -85,B 0,C 180,E1 -23696.646,E2 -23696.646} C_VEL
LIN {X 0,Y 157.263,Z 183.892,A -85,B 0,C 180,E1 -23702.428,E2 -23702.428} C_VEL
LIN {X 0,Y 157.256,Z 183.895,A -85,B 0,C 180,E1 -23706.442,E2 -23706.442} C_VEL
LIN {X 0,Y 157.187,Z 183.898,A -85,B 0,C 180,E1 -23712.115,E2 -23712.115} C_VEL
LIN {X 0,Y 157.186,Z 183.903,A -85,B 0,C 180,E1 -23717.88,E2 -23717.88} C_VEL
LIN {X 0,Y 157.254,Z 183.896,A -85,B 0,C 180,E1 -23723.554,E2 -23723.554} C_VEL
LIN {X 0,Y 157.275,Z 183.89,A -85,B 0,C 180,E1 -23728.102,E2 -23728.102} C_VEL
LIN {X 0,Y 157.304,Z 183.889,A -85,B 0,C 180,E1 -23733.462,E2 -23733.462} C_VEL
LIN {X 0,Y 157.354,Z 183.882,A -85,B 0,C 180,E1 -23739.701,E2 -23739.701} C_VEL
LIN {X 0,Y 157.4,Z 183.874,A -85,B 0,C 180,E1 -23744.46,E2 -23744.46} C_VEL
LIN {X 0,Y 157.681,Z 183.843,A -85,B 0,C 180,E1 -23749.73,E2 -23749.73} C_VEL
LIN {X 0,Y 157.752,Z 183.831,A -85,B 0,C 180,E1 -23752.319,E2 -23752.319} C_VEL
LIN {X 0,Y 158.23,Z 183.774,A -85,B 0,C 180,E1 -23759.999,E2 -23759.999} C_VEL
LIN {X 0,Y 157.75,Z 183.836,A -85,B 0,C 180,E1 -23767.68,E2 -23767.68} C_VEL
LIN {X 0,Y 157.623,Z 183.845,A -85,B 0,C 180,E1 -23771.223,E2 -23771.223} C_VEL
LIN {X 0,Y 157.399,Z 183.88,A -85,B 0,C 180,E1 -23775.539,E2 -23775.539} C_VEL
LIN {X 0,Y 157.296,Z 183.889,A -85,B 0,C 180,E1 -23780.943,E2 -23780.943} C_VEL
LIN {X 0,Y 157.26,Z 183.892,A -85,B 0,C 180,E1 -23786.65,E2 -23786.65} C_VEL
LIN {X 0,Y 157.262,Z 183.895,A -85,B 0,C 180,E1 -23792.43,E2 -23792.43} C_VEL
LIN {X 0,Y 157.252,Z 183.889,A -85,B 0,C 180,E1 -23796.445,E2 -23796.445} C_VEL
LIN {X 0,Y 157.184,Z 183.903,A -85,B 0,C 180,E1 -23802.119,E2 -23802.119} C_VEL
LIN {X 0,Y 157.188,Z 183.905,A -85,B 0,C 180,E1 -23807.885,E2 -23807.885} C_VEL
LIN {X 0,Y 157.348,Z 184.035,A -85,B 0,C 180,E1 -23811.691,E2 -23811.691} C_VEL
LIN {X 0,Y 157.666,Z 185.284,A -85,B 0,C 180,E1 -23812.418,E2 -23812.418} C_VEL
LIN {X 0,Y 165.668,Z 210.745,A -85,B 0,C 180,E1 -23815.145,E2 -23815.145} C_VEL
LIN {X 0,Y 168.383,Z 220.195,A -85,B 0,C 180,E1 -23816.052,E2 -23816.052} C_VEL
LIN {X 0,Y 170.309,Z 240.964,A -85,B 0,C 180,E1 -23817.56,E2 -23817.56} C_VEL
LIN {X 0,Y 167.062,Z 293.98,A -85,B 0,C 180,E1 -23820.638,E2 -23820.638} C_VEL
LIN {X 0,Y 165.76,Z 307.351,A -85,B 0,C 180,E1 -23821.859,E2 -23821.859} C_VEL
LIN {X 0,Y 164.312,Z 318.844,A -85,B 0,C 180,E1 -23823.316,E2 -23823.316} C_VEL
LIN {X 0,Y 162.458,Z 331.336,A -85,B 0,C 180,E1 -23825.422,E2 -23825.422} C_VEL
LIN {X 0,Y 160.421,Z 343.687,A -85,B 0,C 180,E1 -23828.14,E2 -23828.14} C_VEL
LIN {X 0,Y 158.58,Z 354.651,A -85,B 0,C 180,E1 -23831.26,E2 -23831.26} C_VEL
LIN {X 0,Y 157.155,Z 363.595,A -85,B 0,C 180,E1 -23834.438,E2 -23834.438} C_VEL
LIN {X 0,Y 155.99,Z 372.306,A -85,B 0,C 180,E1 -23838.305,E2 -23838.305} C_VEL
LIN {X 0,Y 155.383,Z 378.936,A -85,B 0,C 180,E1 -23842.011,E2 -23842.011} C_VEL
LIN {X 0,Y 154.623,Z 381.753,A -85,B 0,C 180,E1 -23843.916,E2 -23843.916} C_VEL
LIN {X 0,Y 153.028,Z 384.128,A -85,B 0,C 180,E1 -23845.854,E2 -23845.854} C_VEL
LIN {X 0,Y 149.303,Z 388.023,A -85,B 0,C 180,E1 -23849.934,E2 -23849.934} C_VEL
LIN {X 0,Y 148.004,Z 390.258,A -85,B 0,C 180,E1 -23852.864,E2 -23852.864} C_VEL
LIN {X 0,Y 148.064,Z 393.365,A -85,B 0,C 180,E1 -23858.189,E2 -23858.189} C_VEL
LIN {X 0,Y 149.374,Z 394.976,A -85,B 0,C 180,E1 -23863.609,E2 -23863.609} C_VEL
LIN {X 0,Y 151.905,Z 395.121,A -85,B 0,C 180,E1 -23868.899,E2 -23868.899} C_VEL
LIN {X 0,Y 156.059,Z 393.847,A -85,B 0,C 180,E1 -23873.913,E2 -23873.913} C_VEL
LIN {X 0,Y 161.407,Z 391.057,A -85,B 0,C 180,E1 -23878.62,E2 -23878.62} C_VEL
LIN {X 0,Y 167.737,Z 386.724,A -85,B 0,C 180,E1 -23883.005,E2 -23883.005} C_VEL
LIN {X 0,Y 173.309,Z 382.377,A -85,B 0,C 180,E1 -23886.018,E2 -23886.018} C_VEL
LIN {X 0,Y 180.56,Z 375.94,A -85,B 0,C 180,E1 -23889.237,E2 -23889.237} C_VEL
LIN {X 0,Y 188.469,Z 367.714,A -85,B 0,C 180,E1 -23892.163,E2 -23892.163} C_VEL
LIN {X 0,Y 195.704,Z 359.099,A -85,B 0,C 180,E1 -23894.451,E2 -23894.451} C_VEL
LIN {X 0,Y 202.043,Z 350.396,A -85,B 0,C 180,E1 -23896.204,E2 -23896.204} C_VEL
LIN {X 0,Y 208.586,Z 339.846,A -85,B 0,C 180,E1 -23897.841,E2 -23897.841} C_VEL
LIN {X 0,Y 214.794,Z 328.149,A -85,B 0,C 180,E1 -23899.173,E2 -23899.173} C_VEL
LIN {X 0,Y 219.817,Z 316.751,A -85,B 0,C 180,E1 -23900.117,E2 -23900.117} C_VEL
LIN {X 0,Y 224.522,Z 302.879,A -85,B 0,C 180,E1 -23900.994,E2 -23900.994} C_VEL
LIN {X 0,Y 227.858,Z 289.381,A -85,B 0,C 180,E1 -23901.592,E2 -23901.592} C_VEL
LIN {X 0,Y 229.488,Z 279.695,A -85,B 0,C 180,E1 -23902.015,E2 -23902.015} C_VEL
LIN {X 0,Y 228.847,Z 276.734,A -85,B 0,C 180,E1 -23903.728,E2 -23903.728} C_VEL
LIN {X 0,Y 228.436,Z 274.912,A -85,B 0,C 180,E1 -23905.119,E2 -23905.119} C_VEL
LIN {X 0,Y 228.035,Z 272.977,A -85,B 0,C 180,E1 -23907.513,E2 -23907.513} C_VEL
LIN {X 0,Y 227.982,Z 272.515,A -85,B 0,C 180,E1 -23908.395,E2 -23908.395} C_VEL
LIN {X 0,Y 228.202,Z 272.616,A -85,B 0,C 180,E1 -23911.523,E2 -23911.523} C_VEL
LIN {X 0,Y 229.081,Z 274.368,A -85,B 0,C 180,E1 -23914.458,E2 -23914.458} C_VEL
LIN {X 0,Y 229.909,Z 276.74,A -85,B 0,C 180,E1 -23916.377,E2 -23916.377} C_VEL
LIN {X 0,Y 226.944,Z 292.436,A -85,B 0,C 180,E1 -23916.991,E2 -23916.991} C_VEL
LIN {X 0,Y 223.422,Z 305.067,A -85,B 0,C 180,E1 -23917.692,E2 -23917.692} C_VEL
LIN {X 0,Y 218.819,Z 317.583,A -85,B 0,C 180,E1 -23918.661,E2 -23918.661} C_VEL
LIN {X 0,Y 213.814,Z 328.545,A -85,B 0,C 180,E1 -23919.81,E2 -23919.81} C_VEL
LIN {X 0,Y 207.769,Z 339.444,A -85,B 0,C 180,E1 -23921.29,E2 -23921.29} C_VEL
LIN {X 0,Y 200.744,Z 350.18,A -85,B 0,C 180,E1 -23923.212,E2 -23923.212} C_VEL
LIN {X 0,Y 193.972,Z 358.926,A -85,B 0,C 180,E1 -23925.308,E2 -23925.308} C_VEL
LIN {X 0,Y 187.026,Z 366.582,A -85,B 0,C 180,E1 -23927.7,E2 -23927.7} C_VEL
LIN {X 0,Y 180.199,Z 373.197,A -85,B 0,C 180,E1 -23930.459,E2 -23930.459} C_VEL
LIN {X 0,Y 174.501,Z 377.916,A -85,B 0,C 180,E1 -23933.061,E2 -23933.061} C_VEL
LIN {X 0,Y 169.076,Z 381.873,A -85,B 0,C 180,E1 -23936.065,E2 -23936.065} C_VEL
LIN {X 0,Y 163.084,Z 385.481,A -85,B 0,C 180,E1 -23940.001,E2 -23940.001} C_VEL
LIN {X 0,Y 159.905,Z 387.023,A -85,B 0,C 180,E1 -23942.52,E2 -23942.52} C_VEL
LIN {X 0,Y 155.667,Z 388.456,A -85,B 0,C 180,E1 -23946.645,E2 -23946.645} C_VEL
LIN {X 0,Y 152.572,Z 388.803,A -85,B 0,C 180,E1 -23950.618,E2 -23950.618} C_VEL
LIN {X 0,Y 150.843,Z 388.487,A -85,B 0,C 180,E1 -23953.472,E2 -23953.472} C_VEL
LIN {X 0,Y 148.58,Z 386.706,A -85,B 0,C 180,E1 -23958.905,E2 -23958.905} C_VEL
LIN {X 0,Y 147.717,Z 384.773,A -85,B 0,C 180,E1 -23962.373,E2 -23962.373} C_VEL
LIN {X 0,Y 147.337,Z 381.184,A -85,B 0,C 180,E1 -23966.947,E2 -23966.947} C_VEL
LIN {X 0,Y 147.568,Z 376.199,A -85,B 0,C 180,E1 -23971.594,E2 -23971.594} C_VEL
LIN {X 0,Y 148.122,Z 370.776,A -85,B 0,C 180,E1 -23975.509,E2 -23975.509} C_VEL
LIN {X 0,Y 148.95,Z 363.768,A -85,B 0,C 180,E1 -23979.553,E2 -23979.553} C_VEL
LIN {X 0,Y 150.281,Z 354.88,A -85,B 0,C 180,E1 -23983.615,E2 -23983.615} C_VEL
LIN {X 0,Y 151.899,Z 345.228,A -85,B 0,C 180,E1 -23987.127,E2 -23987.127} C_VEL
LIN {X 0,Y 153.621,Z 334.746,A -85,B 0,C 180,E1 -23990.169,E2 -23990.169} C_VEL
LIN {X 0,Y 155.546,Z 323.297,A -85,B 0,C 180,E1 -23992.784,E2 -23992.784} C_VEL
LIN {X 0,Y 157.507,Z 310.499,A -85,B 0,C 180,E1 -23995.051,E2 -23995.051} C_VEL
LIN {X 0,Y 159.091,Z 297.032,A -85,B 0,C 180,E1 -23996.807,E2 -23996.807} C_VEL
LIN {X 0,Y 160.239,Z 283.814,A -85,B 0,C 180,E1 -23998.022,E2 -23998.022} C_VEL
LIN {X 0,Y 164.224,Z 224.078,A -85,B 0,C 180,E1 -24001.571,E2 -24001.571} C_VEL
LIN {X 0,Y 158.943,Z 207.393,A -85,B 0,C 180,E1 -24003.313,E2 -24003.313} C_VEL
LIN {X 0,Y 150.349,Z 185.392,A -85,B 0,C 180,E1 -24006.038,E2 -24006.038} C_VEL
LIN {X 0,Y 150.229,Z 184.772,A -85,B 0,C 180,E1 -24006.201,E2 -24006.201} C_VEL
LIN {X 0,Y 150.303,Z 184.763,A -85,B 0,C 180,E1 -24010.892,E2 -24010.892} C_VEL
LIN {X 0,Y 150.407,Z 184.751,A -85,B 0,C 180,E1 -24016.487,E2 -24016.487} C_VEL
LIN {X 0,Y 150.61,Z 184.725,A -85,B 0,C 180,E1 -24019.24,E2 -24019.24} C_VEL
LIN {X 0,Y 150.702,Z 184.715,A -85,B 0,C 180,E1 -24021.955,E2 -24021.955} C_VEL
LIN {X 0,Y 151.2,Z 184.646,A -85,B 0,C 180,E1 -24029.998,E2 -24029.998} C_VEL
LIN {X 0,Y 150.682,Z 184.71,A -85,B 0,C 180,E1 -24038.041,E2 -24038.041} C_VEL
LIN {X 0,Y 150.574,Z 184.728,A -85,B 0,C 180,E1 -24041.425,E2 -24041.425} C_VEL
LIN {X 0,Y 150.312,Z 184.755,A -85,B 0,C 180,E1 -24046.29,E2 -24046.29} C_VEL
LIN {X 0,Y 150.282,Z 184.764,A -85,B 0,C 180,E1 -24050.719,E2 -24050.719} C_VEL
LIN {X 0,Y 150.184,Z 184.776,A -85,B 0,C 180,E1 -24057.234,E2 -24057.234} C_VEL
LIN {X 0,Y 150.204,Z 184.772,A -85,B 0,C 180,E1 -24062.623,E2 -24062.623} C_VEL
LIN {X 0,Y 150.167,Z 184.779,A -85,B 0,C 180,E1 -24067.472,E2 -24067.472} C_VEL
LIN {X 0,Y 150.13,Z 184.778,A -85,B 0,C 180,E1 -24071.494,E2 -24071.494} C_VEL
LIN {X 0,Y 150.123,Z 184.785,A -85,B 0,C 180,E1 -24075.393,E2 -24075.393} C_VEL
LIN {X 0,Y 150.133,Z 184.78,A -85,B 0,C 180,E1 -24079.052,E2 -24079.052} C_VEL
LIN {X 0,Y 150.171,Z 184.778,A -85,B 0,C 180,E1 -24082.708,E2 -24082.708} C_VEL
LIN {X 0,Y 150.201,Z 184.771,A -85,B 0,C 180,E1 -24087.372,E2 -24087.372} C_VEL
LIN {X 0,Y 150.223,Z 184.773,A -85,B 0,C 180,E1 -24092.729,E2 -24092.729} C_VEL
LIN {X 0,Y 150.278,Z 184.764,A -85,B 0,C 180,E1 -24099.275,E2 -24099.275} C_VEL
LIN {X 0,Y 150.306,Z 184.76,A -85,B 0,C 180,E1 -24103.706,E2 -24103.706} C_VEL
LIN {X 0,Y 150.6,Z 184.725,A -85,B 0,C 180,E1 -24109.241,E2 -24109.241} C_VEL
LIN {X 0,Y 150.691,Z 184.713,A -85,B 0,C 180,E1 -24111.956,E2 -24111.956} C_VEL
LIN {X 0,Y 151.19,Z 184.651,A -85,B 0,C 180,E1 -24119.999,E2 -24119.999} C_VEL
LIN {X 0,Y 150.673,Z 184.715,A -85,B 0,C 180,E1 -24128.043,E2 -24128.043} C_VEL
LIN {X 0,Y 150.566,Z 184.724,A -85,B 0,C 180,E1 -24131.427,E2 -24131.427} C_VEL
LIN {X 0,Y 150.304,Z 184.761,A -85,B 0,C 180,E1 -24136.293,E2 -24136.293} C_VEL
LIN {X 0,Y 150.275,Z 184.763,A -85,B 0,C 180,E1 -24140.722,E2 -24140.722} C_VEL
LIN {X 0,Y 150.178,Z 184.773,A -85,B 0,C 180,E1 -24147.238,E2 -24147.238} C_VEL
LIN {X 0,Y 150.202,Z 184.774,A -85,B 0,C 180,E1 -24152.629,E2 -24152.629} C_VEL
LIN {X 0,Y 150.163,Z 184.776,A -85,B 0,C 180,E1 -24157.476,E2 -24157.476} C_VEL
LIN {X 0,Y 150.127,Z 184.783,A -85,B 0,C 180,E1 -24161.498,E2 -24161.498} C_VEL
LIN {X 0,Y 150.121,Z 184.787,A -85,B 0,C 180,E1 -24165.397,E2 -24165.397} C_VEL
LIN {X 0,Y 150.29,Z 184.924,A -85,B 0,C 180,E1 -24171.281,E2 -24171.281} C_VEL
LIN {X 0,Y 157.249,Z 206.667,A -85,B 0,C 180,E1 -24173.844,E2 -24173.844} C_VEL
LIN {X 0,Y 161.718,Z 222.306,A -85,B 0,C 180,E1 -24175.448,E2 -24175.448} C_VEL
LIN {X 0,Y 163.5,Z 241.356,A -85,B 0,C 180,E1 -24176.896,E2 -24176.896} C_VEL
LIN {X 0,Y 160.087,Z 294.502,A -85,B 0,C 180,E1 -24180.135,E2 -24180.135} C_VEL
LIN {X 0,Y 158.769,Z 307.675,A -85,B 0,C 180,E1 -24181.407,E2 -24181.407} C_VEL
LIN {X 0,Y 157.112,Z 320.011,A -85,B 0,C 180,E1 -24183.072,E2 -24183.072} C_VEL
LIN {X 0,Y 155.188,Z 332.644,A -85,B 0,C 180,E1 -24185.371,E2 -24185.371} C_VEL
LIN {X 0,Y 153.196,Z 344.307,A -85,B 0,C 180,E1 -24188.118,E2 -24188.118} C_VEL
LIN {X 0,Y 151.519,Z 354.138,A -85,B 0,C 180,E1 -24191.056,E2 -24191.056} C_VEL
LIN {X 0,Y 150.066,Z 363.132,A -85,B 0,C 180,E1 -24194.381,E2 -24194.381} C_VEL
LIN {X 0,Y 149.029,Z 370.546,A -85,B 0,C 180,E1 -24197.75,E2 -24197.75} C_VEL
LIN {X 0,Y 148.352,Z 377.788,A -85,B 0,C 180,E1 -24201.832,E2 -24201.832} C_VEL
LIN {X 0,Y 148.158,Z 384.117,A -85,B 0,C 180,E1 -24206.443,E2 -24206.443} C_VEL
LIN {X 0,Y 148.151,Z 387.907,A -85,B 0,C 180,E1 -24210.002,E2 -24210.002} C_VEL
LIN {X 0,Y 148.004,Z 390.258,A -85,B 0,C 180,E1 -24212.864,E2 -24212.864} C_VEL
LIN {X 0,Y 147.217,Z 391.67,A -85,B 0,C 180,E1 -24215.069,E2 -24215.069} C_VEL
LIN {X 0,Y 144.622,Z 393.295,A -85,B 0,C 180,E1 -24218.774,E2 -24218.774} C_VEL
LIN {X 0,Y 142.844,Z 394.111,A -85,B 0,C 180,E1 -24221.854,E2 -24221.854} C_VEL
LIN {X 0,Y 142.546,Z 394.546,A -85,B 0,C 180,E1 -24224.228,E2 -24224.228} C_VEL
LIN {X 0,Y 142.756,Z 394.657,A -85,B 0,C 180,E1 -24225.017,E2 -24225.017} C_VEL
LIN {X 0,Y 145.192,Z 394.976,A -85,B 0,C 180,E1 -24229.808,E2 -24229.808} C_VEL
LIN {X 0,Y 149.598,Z 393.947,A -85,B 0,C 180,E1 -24235.015,E2 -24235.015} C_VEL
LIN {X 0,Y 155.219,Z 391.481,A -85,B 0,C 180,E1 -24239.874,E2 -24239.874} C_VEL
LIN {X 0,Y 160.643,Z 388.335,A -85,B 0,C 180,E1 -24243.592,E2 -24243.592} C_VEL
LIN {X 0,Y 167.689,Z 383.457,A -85,B 0,C 180,E1 -24247.426,E2 -24247.426} C_VEL
LIN {X 0,Y 174.102,Z 378.34,A -85,B 0,C 180,E1 -24250.234,E2 -24250.234} C_VEL
LIN {X 0,Y 182.225,Z 370.894,A -85,B 0,C 180,E1 -24253.205,E2 -24253.205} C_VEL
LIN {X 0,Y 189.614,Z 363.005,A -85,B 0,C 180,E1 -24255.523,E2 -24255.523} C_VEL
LIN {X 0,Y 197.388,Z 353.374,A -85,B 0,C 180,E1 -24257.632,E2 -24257.632} C_VEL
LIN {X 0,Y 204.878,Z 342.457,A -85,B 0,C 180,E1 -24259.413,E2 -24259.413} C_VEL
LIN {X 0,Y 211.065,Z 331.809,A -85,B 0,C 180,E1 -24260.685,E2 -24260.685} C_VEL
LIN {X 0,Y 216.26,Z 321.099,A -85,B 0,C 180,E1 -24261.63,E2 -24261.63} C_VEL
LIN {X 0,Y 221.409,Z 307.764,A -85,B 0,C 180,E1 -24262.521,E2 -24262.521} C_VEL
LIN {X 0,Y 225.4,Z 294.179,A -85,B 0,C 180,E1 -24263.17,E2 -24263.17} C_VEL
LIN {X 0,Y 227.439,Z 284.339,A -85,B 0,C 180,E1 -24263.598,E2 -24263.598} C_VEL
LIN {X 0,Y 226.909,Z 281.636,A -85,B 0,C 180,E1 -24265.572,E2 -24265.572} C_VEL
LIN {X 0,Y 226.629,Z 279.644,A -85,B 0,C 180,E1 -24268.185,E2 -24268.185} C_VEL
LIN {X 0,Y 226.659,Z 279.381,A -85,B 0,C 180,E1 -24270.257,E2 -24270.257} C_VEL
LIN {X 0,Y 227.029,Z 280.126,A -85,B 0,C 180,E1 -24272.616,E2 -24272.616} C_VEL
LIN {X 0,Y 227.613,Z 281.357,A -85,B 0,C 180,E1 -24274.282,E2 -24274.282} C_VEL
LIN {X 0,Y 227.787,Z 282.057,A -85,B 0,C 180,E1 -24274.821,E2 -24274.821} C_VEL
LIN {X 0,Y 225.128,Z 294.377,A -85,B 0,C 180,E1 -24275.302,E2 -24275.302} C_VEL
LIN {X 0,Y 220.949,Z 307.993,A -85,B 0,C 180,E1 -24276.074,E2 -24276.074} C_VEL
LIN {X 0,Y 216.131,Z 320.086,A -85,B 0,C 180,E1 -24277.033,E2 -24277.033} C_VEL
LIN {X 0,Y 210.525,Z 331.407,A -85,B 0,C 180,E1 -24278.236,E2 -24278.236} C_VEL
LIN {X 0,Y 204.48,Z 341.546,A -85,B 0,C 180,E1 -24279.636,E2 -24279.636} C_VEL
LIN {X 0,Y 197.781,Z 351.055,A -85,B 0,C 180,E1 -24281.349,E2 -24281.349} C_VEL
LIN {X 0,Y 190.677,Z 359.707,A -85,B 0,C 180,E1 -24283.404,E2 -24283.404} C_VEL
LIN {X 0,Y 183.849,Z 366.877,A -85,B 0,C 180,E1 -24285.613,E2 -24285.613} C_VEL
LIN {X 0,Y 176.195,Z 373.778,A -85,B 0,C 180,E1 -24288.496,E2 -24288.496} C_VEL
LIN {X 0,Y 169.008,Z 379.273,A -85,B 0,C 180,E1 -24291.631,E2 -24291.631} C_VEL
LIN {X 0,Y 162.182,Z 383.641,A -85,B 0,C 180,E1 -24295.353,E2 -24295.353} C_VEL
LIN {X 0,Y 158.806,Z 385.42,A -85,B 0,C 180,E1 -24297.464,E2 -24297.464} C_VEL
LIN {X 0,Y 154.628,Z 387.296,A -85,B 0,C 180,E1 -24300.531,E2 -24300.531} C_VEL
LIN {X 0,Y 149.315,Z 388.812,A -85,B 0,C 180,E1 -24305.402,E2 -24305.402} C_VEL
LIN {X 0,Y 146.924,Z 389.036,A -85,B 0,C 180,E1 -24308.251,E2 -24308.251} C_VEL
LIN {X 0,Y 144.05,Z 388.547,A -85,B 0,C 180,E1 -24312.628,E2 -24312.628} C_VEL
LIN {X 0,Y 141.96,Z 387.01,A -85,B 0,C 180,E1 -24317.281,E2 -24317.281} C_VEL
LIN {X 0,Y 140.69,Z 384.401,A -85,B 0,C 180,E1 -24322.004,E2 -24322.004} C_VEL
LIN {X 0,Y 140.269,Z 380.627,A -85,B 0,C 180,E1 -24326.804,E2 -24326.804} C_VEL
LIN {X 0,Y 140.514,Z 375.363,A -85,B 0,C 180,E1 -24331.754,E2 -24331.754} C_VEL
LIN {X 0,Y 141.109,Z 369.748,A -85,B 0,C 180,E1 -24335.819,E2 -24335.819} C_VEL
LIN {X 0,Y 141.994,Z 362.417,A -85,B 0,C 180,E1 -24340.05,E2 -24340.05} C_VEL
LIN {X 0,Y 143.417,Z 353.197,A -85,B 0,C 180,E1 -24344.292,E2 -24344.292} C_VEL
LIN {X 0,Y 144.991,Z 344.028,A -85,B 0,C 180,E1 -24347.671,E2 -24347.671} C_VEL
LIN {X 0,Y 146.859,Z 332.862,A -85,B 0,C 180,E1 -24350.945,E2 -24350.945} C_VEL
LIN {X 0,Y 148.721,Z 322.08,A -85,B 0,C 180,E1 -24353.453,E2 -24353.453} C_VEL
LIN {X 0,Y 150.508,Z 310.636,A -85,B 0,C 180,E1 -24355.545,E2 -24355.545} C_VEL
LIN {X 0,Y 152.199,Z 296.79,A -85,B 0,C 180,E1 -24357.43,E2 -24357.43} C_VEL
LIN {X 0,Y 153.434,Z 283.044,A -85,B 0,C 180,E1 -24358.711,E2 -24358.711} C_VEL
LIN {X 0,Y 157.356,Z 225.136,A -85,B 0,C 180,E1 -24362.302,E2 -24362.302} C_VEL
LIN {X 0,Y 152.732,Z 210.416,A -85,B 0,C 180,E1 -24363.92,E2 -24363.92} C_VEL
LIN {X 0,Y 144.897,Z 190.386,A -85,B 0,C 180,E1 -24366.485,E2 -24366.485} C_VEL
LIN {X 0,Y 143.158,Z 185.652,A -85,B 0,C 180,E1 -24367.157,E2 -24367.157} C_VEL
LIN {X 0,Y 143.248,Z 185.642,A -85,B 0,C 180,E1 -24369.911,E2 -24369.911} C_VEL
LIN {X 0,Y 143.308,Z 185.635,A -85,B 0,C 180,E1 -24375.804,E2 -24375.804} C_VEL
LIN {X 0,Y 143.537,Z 185.606,A -85,B 0,C 180,E1 -24378.703,E2 -24378.703} C_VEL
LIN {X 0,Y 143.624,Z 185.594,A -85,B 0,C 180,E1 -24381.556,E2 -24381.556} C_VEL
LIN {X 0,Y 144.159,Z 185.523,A -85,B 0,C 180,E1 -24389.998,E2 -24389.998} C_VEL
LIN {X 0,Y 143.608,Z 185.59,A -85,B 0,C 180,E1 -24398.44,E2 -24398.44} C_VEL
LIN {X 0,Y 143.499,Z 185.611,A -85,B 0,C 180,E1 -24401.611,E2 -24401.611} C_VEL
LIN {X 0,Y 143.252,Z 185.635,A -85,B 0,C 180,E1 -24407.117,E2 -24407.117} C_VEL
LIN {X 0,Y 143.219,Z 185.646,A -85,B 0,C 180,E1 -24411.191,E2 -24411.191} C_VEL
LIN {X 0,Y 143.141,Z 185.654,A -85,B 0,C 180,E1 -24417.897,E2 -24417.897} C_VEL
LIN {X 0,Y 143.134,Z 185.65,A -85,B 0,C 180,E1 -24423.412,E2 -24423.412} C_VEL
LIN {X 0,Y 143.049,Z 185.664,A -85,B 0,C 180,E1 -24429.691,E2 -24429.691} C_VEL
LIN {X 0,Y 143.03,Z 185.666,A -85,B 0,C 180,E1 -24433.461,E2 -24433.461} C_VEL
LIN {X 0,Y 143.034,Z 185.666,A -85,B 0,C 180,E1 -24437.475,E2 -24437.475} C_VEL
LIN {X 0,Y 143.067,Z 185.66,A -85,B 0,C 180,E1 -24441.807,E2 -24441.807} C_VEL
LIN {X 0,Y 143.168,Z 185.647,A -85,B 0,C 180,E1 -24447.317,E2 -24447.317} C_VEL
LIN {X 0,Y 143.171,Z 185.65,A -85,B 0,C 180,E1 -24452.073,E2 -24452.073} C_VEL
LIN {X 0,Y 143.216,Z 185.644,A -85,B 0,C 180,E1 -24458.802,E2 -24458.802} C_VEL
LIN {X 0,Y 143.246,Z 185.64,A -85,B 0,C 180,E1 -24462.879,E2 -24462.879} C_VEL
LIN {X 0,Y 143.526,Z 185.606,A -85,B 0,C 180,E1 -24468.704,E2 -24468.704} C_VEL
LIN {X 0,Y 143.613,Z 185.595,A -85,B 0,C 180,E1 -24471.557,E2 -24471.557} C_VEL
LIN {X 0,Y 144.149,Z 185.528,A -85,B 0,C 180,E1 -24479.999,E2 -24479.999} C_VEL
LIN {X 0,Y 143.599,Z 185.595,A -85,B 0,C 180,E1 -24488.442,E2 -24488.442} C_VEL
LIN {X 0,Y 143.491,Z 185.606,A -85,B 0,C 180,E1 -24491.613,E2 -24491.613} C_VEL
LIN {X 0,Y 143.245,Z 185.64,A -85,B 0,C 180,E1 -24497.12,E2 -24497.12} C_VEL
LIN {X 0,Y 143.212,Z 185.644,A -85,B 0,C 180,E1 -24501.194,E2 -24501.194} C_VEL
LIN {X 0,Y 143.135,Z 185.651,A -85,B 0,C 180,E1 -24507.901,E2 -24507.901} C_VEL
LIN {X 0,Y 143.132,Z 185.654,A -85,B 0,C 180,E1 -24513.417,E2 -24513.417} C_VEL
LIN {X 0,Y 143.046,Z 185.666,A -85,B 0,C 180,E1 -24519.695,E2 -24519.695} C_VEL
LIN {X 0,Y 143.028,Z 185.669,A -85,B 0,C 180,E1 -24523.465,E2 -24523.465} C_VEL
LIN {X 0,Y 143.204,Z 185.849,A -85,B 0,C 180,E1 -24530.292,E2 -24530.292} C_VEL
LIN {X 0,Y 148.506,Z 201.322,A -85,B 0,C 180,E1 -24532.262,E2 -24532.262} C_VEL
LIN {X 0,Y 155.051,Z 223.77,A -85,B 0,C 180,E1 -24534.745,E2 -24534.745} C_VEL
LIN {X 0,Y 156.609,Z 242.917,A -85,B 0,C 180,E1 -24536.251,E2 -24536.251} C_VEL
LIN {X 0,Y 153.217,Z 294.122,A -85,B 0,C 180,E1 -24539.51,E2 -24539.51} C_VEL
LIN {X 0,Y 151.778,Z 307.986,A -85,B 0,C 180,E1 -24540.912,E2 -24540.912} C_VEL
LIN {X 0,Y 150.097,Z 320.004,A -85,B 0,C 180,E1 -24542.62,E2 -24542.62} C_VEL
LIN {X 0,Y 148.097,Z 332.912,A -85,B 0,C 180,E1 -24545.094,E2 -24545.094} C_VEL
LIN {X 0,Y 146.189,Z 343.662,A -85,B 0,C 180,E1 -24547.756,E2 -24547.756} C_VEL
LIN {X 0,Y 144.473,Z 353.518,A -85,B 0,C 180,E1 -24550.833,E2 -24550.833} C_VEL
LIN {X 0,Y 142.999,Z 362.53,A -85,B 0,C 180,E1 -24554.32,E2 -24554.32} C_VEL
LIN {X 0,Y 141.84,Z 371.347,A -85,B 0,C 180,E1 -24558.571,E2 -24558.571} C_VEL
LIN {X 0,Y 141.251,Z 378.335,A -85,B 0,C 180,E1 -24562.857,E2 -24562.857} C_VEL
LIN {X 0,Y 141.121,Z 383.869,A -85,B 0,C 180,E1 -24567.148,E2 -24567.148} C_VEL
LIN {X 0,Y 141.077,Z 388.101,A -85,B 0,C 180,E1 -24571.43,E2 -24571.43} C_VEL
LIN {X 0,Y 140.866,Z 391.15,A -85,B 0,C 180,E1 -24575.729,E2 -24575.729} C_VEL
LIN {X 0,Y 141.632,Z 393.785,A -85,B 0,C 180,E1 -24581.451,E2 -24581.451} C_VEL
LIN {X 0,Y 142.756,Z 394.657,A -85,B 0,C 180,E1 -24585.017,E2 -24585.017} C_VEL
LIN {X 0,Y 143.15,Z 394.941,A -85,B 0,C 180,E1 -24587.38,E2 -24587.38} C_VEL
LIN {X 0,Y 142.673,Z 394.838,A -85,B 0,C 180,E1 -24591.354,E2 -24591.354} C_VEL
LIN {X 0,Y 143.005,Z 394.236,A -85,B 0,C 180,E1 -24595.31,E2 -24595.31} C_VEL
LIN {X 0,Y 144.615,Z 393.572,A -85,B 0,C 180,E1 -24597.551,E2 -24597.551} C_VEL
LIN {X 0,Y 149.115,Z 391.87,A -85,B 0,C 180,E1 -24601.231,E2 -24601.231} C_VEL
LIN {X 0,Y 156.105,Z 388.237,A -85,B 0,C 180,E1 -24605.825,E2 -24605.825} C_VEL
LIN {X 0,Y 162.171,Z 384.458,A -85,B 0,C 180,E1 -24608.934,E2 -24608.934} C_VEL
LIN {X 0,Y 168.832,Z 379.7,A -85,B 0,C 180,E1 -24611.764,E2 -24611.764} C_VEL
LIN {X 0,Y 177.243,Z 372.704,A -85,B 0,C 180,E1 -24614.737,E2 -24614.737} C_VEL
LIN {X 0,Y 184.889,Z 365.312,A -85,B 0,C 180,E1 -24617.034,E2 -24617.034} C_VEL
LIN {X 0,Y 192.874,Z 356.301,A -85,B 0,C 180,E1 -24619.124,E2 -24619.124} C_VEL
LIN {X 0,Y 201.168,Z 345.223,A -85,B 0,C 180,E1 -24621.019,E2 -24621.019} C_VEL
LIN {X 0,Y 208.857,Z 332.839,A -85,B 0,C 180,E1 -24622.504,E2 -24622.504} C_VEL
LIN {X 0,Y 214.396,Z 322.138,A -85,B 0,C 180,E1 -24623.432,E2 -24623.432} C_VEL
LIN {X 0,Y 219.605,Z 309.6,A -85,B 0,C 180,E1 -24624.252,E2 -24624.252} C_VEL
LIN {X 0,Y 224.105,Z 295.241,A -85,B 0,C 180,E1 -24624.921,E2 -24624.921} C_VEL
LIN {X 0,Y 225.479,Z 289.47,A -85,B 0,C 180,E1 -24625.143,E2 -24625.143} C_VEL
LIN {X 0,Y 225.309,Z 288.172,A -85,B 0,C 180,E1 -24626.214,E2 -24626.214} C_VEL
LIN {X 0,Y 225.202,Z 286.532,A -85,B 0,C 180,E1 -24628.439,E2 -24628.439} C_VEL
LIN {X 0,Y 225.322,Z 286.438,A -85,B 0,C 180,E1 -24630.853,E2 -24630.853} C_VEL
LIN {X 0,Y 225.767,Z 287.44,A -85,B 0,C 180,E1 -24633.182,E2 -24633.182} C_VEL
LIN {X 0,Y 222.216,Z 301.071,A -85,B 0,C 180,E1 -24633.825,E2 -24633.825} C_VEL
LIN {X 0,Y 217.901,Z 313.156,A -85,B 0,C 180,E1 -24634.57,E2 -24634.57} C_VEL
LIN {X 0,Y 212.534,Z 324.996,A -85,B 0,C 180,E1 -24635.585,E2 -24635.585} C_VEL
LIN {X 0,Y 206.449,Z 335.815,A -85,B 0,C 180,E1 -24636.805,E2 -24636.805} C_VEL
LIN {X 0,Y 199.713,Z 345.98,A -85,B 0,C 180,E1 -24638.316,E2 -24638.316} C_VEL
LIN {X 0,Y 192.002,Z 355.759,A -85,B 0,C 180,E1 -24640.233,E2 -24640.233} C_VEL
LIN {X 0,Y 183.448,Z 364.811,A -85,B 0,C 180,E1 -24642.67,E2 -24642.67} C_VEL
LIN {X 0,Y 176.489,Z 371.14,A -85,B 0,C 180,E1 -24644.946,E2 -24644.946} C_VEL
LIN {X 0,Y 168.542,Z 377.328,A -85,B 0,C 180,E1 -24647.966,E2 -24647.966} C_VEL
LIN {X 0,Y 161.326,Z 381.968,A -85,B 0,C 180,E1 -24651.23,E2 -24651.23} C_VEL
LIN {X 0,Y 154.936,Z 385.384,A -85,B 0,C 180,E1 -24654.795,E2 -24654.795} C_VEL
LIN {X 0,Y 151.03,Z 387.042,A -85,B 0,C 180,E1 -24657.333,E2 -24657.333} C_VEL
LIN {X 0,Y 147.494,Z 388.25,A -85,B 0,C 180,E1 -24660.001,E2 -24660.001} C_VEL
LIN {X 0,Y 144.346,Z 388.986,A -85,B 0,C 180,E1 -24662.791,E2 -24662.791} C_VEL
LIN {X 0,Y 141.329,Z 389.275,A -85,B 0,C 180,E1 -24665.958,E2 -24665.958} C_VEL
LIN {X 0,Y 137.234,Z 388.556,A -85,B 0,C 180,E1 -24671.821,E2 -24671.821} C_VEL
LIN {X 0,Y 135.668,Z 387.497,A -85,B 0,C 180,E1 -24675.012,E2 -24675.012} C_VEL
LIN {X 0,Y 134.169,Z 385.356,A -85,B 0,C 180,E1 -24679.453,E2 -24679.453} C_VEL
LIN {X 0,Y 133.271,Z 381.452,A -85,B 0,C 180,E1 -24684.954,E2 -24684.954} C_VEL
LIN {X 0,Y 133.354,Z 376.544,A -85,B 0,C 180,E1 -24690.045,E2 -24690.045} C_VEL
LIN {X 0,Y 133.941,Z 369.948,A -85,B 0,C 180,E1 -24695.253,E2 -24695.253} C_VEL
LIN {X 0,Y 134.815,Z 362.713,A -85,B 0,C 180,E1 -24699.689,E2 -24699.689} C_VEL
LIN {X 0,Y 136.164,Z 353.886,A -85,B 0,C 180,E1 -24703.99,E2 -24703.99} C_VEL
LIN {X 0,Y 137.804,Z 344.426,A -85,B 0,C 180,E1 -24707.69,E2 -24707.69} C_VEL
LIN {X 0,Y 139.76,Z 333.007,A -85,B 0,C 180,E1 -24711.21,E2 -24711.21} C_VEL
LIN {X 0,Y 141.736,Z 321.892,A -85,B 0,C 180,E1 -24713.91,E2 -24713.91} C_VEL
LIN {X 0,Y 143.706,Z 309.397,A -85,B 0,C 180,E1 -24716.244,E2 -24716.244} C_VEL
LIN {X 0,Y 145.317,Z 296.318,A -85,B 0,C 180,E1 -24718.069,E2 -24718.069} C_VEL
LIN {X 0,Y 146.563,Z 282.83,A -85,B 0,C 180,E1 -24719.366,E2 -24719.366} C_VEL
LIN {X 0,Y 150.557,Z 226.34,A -85,B 0,C 180,E1 -24723.055,E2 -24723.055} C_VEL
LIN {X 0,Y 145.921,Z 211.805,A -85,B 0,C 180,E1 -24724.723,E2 -24724.723} C_VEL
LIN {X 0,Y 137.041,Z 189.253,A -85,B 0,C 180,E1 -24727.856,E2 -24727.856} C_VEL
LIN {X 0,Y 136.142,Z 186.528,A -85,B 0,C 180,E1 -24728.315,E2 -24728.315} C_VEL
LIN {X 0,Y 136.168,Z 186.525,A -85,B 0,C 180,E1 -24731.958,E2 -24731.958} C_VEL
LIN {X 0,Y 136.429,Z 186.493,A -85,B 0,C 180,E1 -24738.176,E2 -24738.176} C_VEL
LIN {X 0,Y 136.55,Z 186.475,A -85,B 0,C 180,E1 -24741.115,E2 -24741.115} C_VEL
LIN {X 0,Y 137.115,Z 186.4,A -85,B 0,C 180,E1 -24749.997,E2 -24749.997} C_VEL
LIN {X 0,Y 136.537,Z 186.471,A -85,B 0,C 180,E1 -24758.881,E2 -24758.881} C_VEL
LIN {X 0,Y 136.415,Z 186.493,A -85,B 0,C 180,E1 -24761.89,E2 -24761.89} C_VEL
LIN {X 0,Y 136.165,Z 186.521,A -85,B 0,C 180,E1 -24768.037,E2 -24768.037} C_VEL
LIN {X 0,Y 136.143,Z 186.526,A -85,B 0,C 180,E1 -24771.687,E2 -24771.687} C_VEL
LIN {X 0,Y 136.06,Z 186.536,A -85,B 0,C 180,E1 -24778.583,E2 -24778.583} C_VEL
LIN {X 0,Y 136.038,Z 186.534,A -85,B 0,C 180,E1 -24784.627,E2 -24784.627} C_VEL
LIN {X 0,Y 136.022,Z 186.54,A -85,B 0,C 180,E1 -24789.191,E2 -24789.191} C_VEL
LIN {X 0,Y 135.975,Z 186.545,A -85,B 0,C 180,E1 -24793.646,E2 -24793.646} C_VEL
LIN {X 0,Y 135.979,Z 186.545,A -85,B 0,C 180,E1 -24797.785,E2 -24797.785} C_VEL
LIN {X 0,Y 136.016,Z 186.538,A -85,B 0,C 180,E1 -24801.68,E2 -24801.68} C_VEL
LIN {X 0,Y 136.047,Z 186.537,A -85,B 0,C 180,E1 -24805.74,E2 -24805.74} C_VEL
LIN {X 0,Y 136.112,Z 186.53,A -85,B 0,C 180,E1 -24812.308,E2 -24812.308} C_VEL
LIN {X 0,Y 136.179,Z 186.521,A -85,B 0,C 180,E1 -24818.822,E2 -24818.822} C_VEL
LIN {X 0,Y 136.216,Z 186.511,A -85,B 0,C 180,E1 -24825.049,E2 -24825.049} C_VEL
LIN {X 0,Y 136.419,Z 186.491,A -85,B 0,C 180,E1 -24828.177,E2 -24828.177} C_VEL
LIN {X 0,Y 136.539,Z 186.475,A -85,B 0,C 180,E1 -24831.116,E2 -24831.116} C_VEL
LIN {X 0,Y 137.106,Z 186.405,A -85,B 0,C 180,E1 -24839.999,E2 -24839.999} C_VEL
LIN {X 0,Y 136.528,Z 186.476,A -85,B 0,C 180,E1 -24848.883,E2 -24848.883} C_VEL
LIN {X 0,Y 136.407,Z 186.49,A -85,B 0,C 180,E1 -24851.893,E2 -24851.893} C_VEL
LIN {X 0,Y 136.157,Z 186.519,A -85,B 0,C 180,E1 -24858.041,E2 -24858.041} C_VEL
LIN {X 0,Y 136.136,Z 186.527,A -85,B 0,C 180,E1 -24861.69,E2 -24861.69} C_VEL
LIN {X 0,Y 136.055,Z 186.533,A -85,B 0,C 180,E1 -24868.587,E2 -24868.587} C_VEL
LIN {X 0,Y 136.034,Z 186.537,A -85,B 0,C 180,E1 -24874.631,E2 -24874.631} C_VEL
LIN {X 0,Y 136.018,Z 186.542,A -85,B 0,C 180,E1 -24879.196,E2 -24879.196} C_VEL
LIN {X 0,Y 135.972,Z 186.548,A -85,B 0,C 180,E1 -24883.65,E2 -24883.65} C_VEL
LIN {X 0,Y 136.039,Z 186.541,A -85,B 0,C 180,E1 -24889.137,E2 -24889.137} C_VEL
LIN {X 0,Y 137.889,Z 191.337,A -85,B 0,C 180,E1 -24889.864,E2 -24889.864} C_VEL
LIN {X 0,Y 142.159,Z 203.882,A -85,B 0,C 180,E1 -24891.535,E2 -24891.535} C_VEL
LIN {X 0,Y 148.308,Z 224.746,A -85,B 0,C 180,E1 -24893.955,E2 -24893.955} C_VEL
LIN {X 0,Y 149.817,Z 243.345,A -85,B 0,C 180,E1 -24895.489,E2 -24895.489} C_VEL
LIN {X 0,Y 146.38,Z 293.357,A -85,B 0,C 180,E1 -24898.83,E2 -24898.83} C_VEL
LIN {X 0,Y 144.824,Z 307.932,A -85,B 0,C 180,E1 -24900.374,E2 -24900.374} C_VEL
LIN {X 0,Y 142.957,Z 320.745,A -85,B 0,C 180,E1 -24902.324,E2 -24902.324} C_VEL
LIN {X 0,Y 141.188,Z 331.915,A -85,B 0,C 180,E1 -24904.578,E2 -24904.578} C_VEL
LIN {X 0,Y 139.233,Z 342.815,A -85,B 0,C 180,E1 -24907.366,E2 -24907.366} C_VEL
LIN {X 0,Y 137.452,Z 352.803,A -85,B 0,C 180,E1 -24910.591,E2 -24910.591} C_VEL
LIN {X 0,Y 135.934,Z 361.891,A -85,B 0,C 180,E1 -24914.253,E2 -24914.253} C_VEL
LIN {X 0,Y 134.772,Z 370.789,A -85,B 0,C 180,E1 -24918.726,E2 -24918.726} C_VEL
LIN {X 0,Y 134.216,Z 377.856,A -85,B 0,C 180,E1 -24923.236,E2 -24923.236} C_VEL
LIN {X 0,Y 134.089,Z 382.588,A -85,B 0,C 180,E1 -24926.998,E2 -24926.998} C_VEL
LIN {X 0,Y 134.071,Z 387.026,A -85,B 0,C 180,E1 -24931.504,E2 -24931.504} C_VEL
LIN {X 0,Y 133.857,Z 390.266,A -85,B 0,C 180,E1 -24936.03,E2 -24936.03} C_VEL
LIN {X 0,Y 134.08,Z 391.931,A -85,B 0,C 180,E1 -24939.05,E2 -24939.05} C_VEL
LIN {X 0,Y 135.618,Z 394.054,A -85,B 0,C 180,E1 -24945.02,E2 -24945.02} C_VEL
LIN {X 0,Y 138.525,Z 394.743,A -85,B 0,C 180,E1 -24950.805,E2 -24950.805} C_VEL
LIN {X 0,Y 143.184,Z 394.039,A -85,B 0,C 180,E1 -24956.218,E2 -24956.218} C_VEL
LIN {X 0,Y 144.615,Z 393.572,A -85,B 0,C 180,E1 -24957.551,E2 -24957.551} C_VEL
LIN {X 0,Y 146.452,Z 392.785,A -85,B 0,C 180,E1 -24959.741,E2 -24959.741} C_VEL
LIN {X 0,Y 148.261,Z 391.197,A -85,B 0,C 180,E1 -24963.488,E2 -24963.488} C_VEL
LIN {X 0,Y 150.686,Z 389.05,A -85,B 0,C 180,E1 -24967.071,E2 -24967.071} C_VEL
LIN {X 0,Y 153.389,Z 387.37,A -85,B 0,C 180,E1 -24968.937,E2 -24968.937} C_VEL
LIN {X 0,Y 161.327,Z 382.6,A -85,B 0,C 180,E1 -24972.475,E2 -24972.475} C_VEL
LIN {X 0,Y 171.12,Z 375.504,A -85,B 0,C 180,E1 -24975.953,E2 -24975.953} C_VEL
LIN {X 0,Y 178.935,Z 368.804,A -85,B 0,C 180,E1 -24978.27,E2 -24978.27} C_VEL
LIN {X 0,Y 187.068,Z 360.617,A -85,B 0,C 180,E1 -24980.371,E2 -24980.371} C_VEL
LIN {X 0,Y 195.55,Z 350.66,A -85,B 0,C 180,E1 -24982.251,E2 -24982.251} C_VEL
LIN {X 0,Y 202.722,Z 340.761,A -85,B 0,C 180,E1 -24983.633,E2 -24983.633} C_VEL
LIN {X 0,Y 209.657,Z 329.253,A -85,B 0,C 180,E1 -24984.796,E2 -24984.796} C_VEL
LIN {X 0,Y 215.773,Z 316.793,A -85,B 0,C 180,E1 -24985.678,E2 -24985.678} C_VEL
LIN {X 0,Y 220.327,Z 305.168,A -85,B 0,C 180,E1 -24986.329,E2 -24986.329} C_VEL
LIN {X 0,Y 223.533,Z 294.689,A -85,B 0,C 180,E1 -24986.79,E2 -24986.79} C_VEL
LIN {X 0,Y 223.533,Z 293.399,A -85,B 0,C 180,E1 -24988.581,E2 -24988.581} C_VEL
LIN {X 0,Y 223.708,Z 293.418,A -85,B 0,C 180,E1 -24991.281,E2 -24991.281} C_VEL
LIN {X 0,Y 223.738,Z 293.583,A -85,B 0,C 180,E1 -24991.63,E2 -24991.63} C_VEL
LIN {X 0,Y 219.81,Z 306.126,A -85,B 0,C 180,E1 -24992.248,E2 -24992.248} C_VEL
LIN {X 0,Y 214.694,Z 318.553,A -85,B 0,C 180,E1 -24993.081,E2 -24993.081} C_VEL
LIN {X 0,Y 209.073,Z 329.626,A -85,B 0,C 180,E1 -24994.088,E2 -24994.088} C_VEL
LIN {X 0,Y 201.771,Z 341.227,A -85,B 0,C 180,E1 -24995.47,E2 -24995.47} C_VEL
LIN {X 0,Y 194.242,Z 351.197,A -85,B 0,C 180,E1 -24997.111,E2 -24997.111} C_VEL
LIN {X 0,Y 186.405,Z 359.946,A -85,B 0,C 180,E1 -24999.011,E2 -24999.011} C_VEL
LIN {X 0,Y 177.359,Z 368.473,A -85,B 0,C 180,E1 -25001.518,E2 -25001.518} C_VEL
LIN {X 0,Y 169.559,Z 374.659,A -85,B 0,C 180,E1 -25004.073,E2 -25004.073} C_VEL
LIN {X 0,Y 160.879,Z 380.403,A -85,B 0,C 180,E1 -25007.384,E2 -25007.384} C_VEL
LIN {X 0,Y 153.662,Z 384.315,A -85,B 0,C 180,E1 -25010.789,E2 -25010.789} C_VEL
LIN {X 0,Y 147.14,Z 387.075,A -85,B 0,C 180,E1 -25014.519,E2 -25014.519} C_VEL
LIN {X 0,Y 140.578,Z 388.972,A -85,B 0,C 180,E1 -25019.229,E2 -25019.229} C_VEL
LIN {X 0,Y 136.524,Z 389.508,A -85,B 0,C 180,E1 -25022.951,E2 -25022.951} C_VEL
LIN {X 0,Y 133.793,Z 389.421,A -85,B 0,C 180,E1 -25026.031,E2 -25026.031} C_VEL
LIN {X 0,Y 131.467,Z 388.917,A -85,B 0,C 180,E1 -25029.229,E2 -25029.229} C_VEL
LIN {X 0,Y 129.596,Z 387.961,A -85,B 0,C 180,E1 -25032.529,E2 -25032.529} C_VEL
LIN {X 0,Y 128.113,Z 386.525,A -85,B 0,C 180,E1 -25035.921,E2 -25035.921} C_VEL
LIN {X 0,Y 126.654,Z 383.463,A -85,B 0,C 180,E1 -25041.191,E2 -25041.191} C_VEL
LIN {X 0,Y 126.186,Z 378.813,A -85,B 0,C 180,E1 -25046.979,E2 -25046.979} C_VEL
LIN {X 0,Y 126.443,Z 373.622,A -85,B 0,C 180,E1 -25051.849,E2 -25051.849} C_VEL
LIN {X 0,Y 127.079,Z 367.4,A -85,B 0,C 180,E1 -25056.48,E2 -25056.48} C_VEL
LIN {X 0,Y 128.121,Z 359.479,A -85,B 0,C 180,E1 -25061.168,E2 -25061.168} C_VEL
LIN {X 0,Y 129.465,Z 351.23,A -85,B 0,C 180,E1 -25065.11,E2 -25065.11} C_VEL
LIN {X 0,Y 131.284,Z 341.017,A -85,B 0,C 180,E1 -25069.046,E2 -25069.046} C_VEL
LIN {X 0,Y 133.198,Z 330.218,A -85,B 0,C 180,E1 -25072.323,E2 -25072.323} C_VEL
LIN {X 0,Y 135.307,Z 318.237,A -85,B 0,C 180,E1 -25075.153,E2 -25075.153} C_VEL
LIN {X 0,Y 137.217,Z 306.145,A -85,B 0,C 180,E1 -25077.343,E2 -25077.343} C_VEL
LIN {X 0,Y 138.707,Z 292.817,A -85,B 0,C 180,E1 -25079.116,E2 -25079.116} C_VEL
LIN {X 0,Y 140.026,Z 278.529,A -85,B 0,C 180,E1 -25080.378,E2 -25080.378} C_VEL
LIN {X 0,Y 143.756,Z 228.039,A -85,B 0,C 180,E1 -25083.792,E2 -25083.792} C_VEL
LIN {X 0,Y 140.209,Z 216.166,A -85,B 0,C 180,E1 -25085.205,E2 -25085.205} C_VEL
LIN {X 0,Y 131.928,Z 194.764,A -85,B 0,C 180,E1 -25088.279,E2 -25088.279} C_VEL
LIN {X 0,Y 129.145,Z 187.671,A -85,B 0,C 180,E1 -25089.386,E2 -25089.386} C_VEL
LIN {X 0,Y 129.108,Z 187.403,A -85,B 0,C 180,E1 -25089.692,E2 -25089.692} C_VEL
LIN {X 0,Y 129.149,Z 187.4,A -85,B 0,C 180,E1 -25094.209,E2 -25094.209} C_VEL
LIN {X 0,Y 129.347,Z 187.374,A -85,B 0,C 180,E1 -25097.97,E2 -25097.97} C_VEL
LIN {X 0,Y 129.473,Z 187.357,A -85,B 0,C 180,E1 -25100.625,E2 -25100.625} C_VEL
LIN {X 0,Y 130.071,Z 187.277,A -85,B 0,C 180,E1 -25109.997,E2 -25109.997} C_VEL
LIN {X 0,Y 129.463,Z 187.353,A -85,B 0,C 180,E1 -25119.37,E2 -25119.37} C_VEL
LIN {X 0,Y 129.298,Z 187.378,A -85,B 0,C 180,E1 -25122.555,E2 -25122.555} C_VEL
LIN {X 0,Y 129.081,Z 187.404,A -85,B 0,C 180,E1 -25129.064,E2 -25129.064} C_VEL
LIN {X 0,Y 129.034,Z 187.411,A -85,B 0,C 180,E1 -25132.409,E2 -25132.409} C_VEL
LIN {X 0,Y 128.998,Z 187.417,A -85,B 0,C 180,E1 -25139.359,E2 -25139.359} C_VEL
LIN {X 0,Y 128.954,Z 187.419,A -85,B 0,C 180,E1 -25145.163,E2 -25145.163} C_VEL
LIN {X 0,Y 128.92,Z 187.421,A -85,B 0,C 180,E1 -25150.853,E2 -25150.853} C_VEL
LIN {X 0,Y 128.908,Z 187.428,A -85,B 0,C 180,E1 -25155.129,E2 -25155.129} C_VEL
LIN {X 0,Y 128.93,Z 187.419,A -85,B 0,C 180,E1 -25159.738,E2 -25159.738} C_VEL
LIN {X 0,Y 128.951,Z 187.423,A -85,B 0,C 180,E1 -25164.832,E2 -25164.832} C_VEL
LIN {X 0,Y 129.012,Z 187.412,A -85,B 0,C 180,E1 -25170.64,E2 -25170.64} C_VEL
LIN {X 0,Y 129.063,Z 187.402,A -85,B 0,C 180,E1 -25177.769,E2 -25177.769} C_VEL
LIN {X 0,Y 129.139,Z 187.395,A -85,B 0,C 180,E1 -25184.209,E2 -25184.209} C_VEL
LIN {X 0,Y 129.337,Z 187.373,A -85,B 0,C 180,E1 -25187.972,E2 -25187.972} C_VEL
LIN {X 0,Y 129.463,Z 187.358,A -85,B 0,C 180,E1 -25190.626,E2 -25190.626} C_VEL
LIN {X 0,Y 130.061,Z 187.282,A -85,B 0,C 180,E1 -25199.999,E2 -25199.999} C_VEL
LIN {X 0,Y 129.454,Z 187.356,A -85,B 0,C 180,E1 -25209.373,E2 -25209.373} C_VEL
LIN {X 0,Y 129.29,Z 187.378,A -85,B 0,C 180,E1 -25212.558,E2 -25212.558} C_VEL
LIN {X 0,Y 129.073,Z 187.401,A -85,B 0,C 180,E1 -25219.068,E2 -25219.068} C_VEL
LIN {X 0,Y 129.027,Z 187.412,A -85,B 0,C 180,E1 -25222.413,E2 -25222.413} C_VEL
LIN {X 0,Y 128.993,Z 187.415,A -85,B 0,C 180,E1 -25229.363,E2 -25229.363} C_VEL
LIN {X 0,Y 128.949,Z 187.416,A -85,B 0,C 180,E1 -25235.167,E2 -25235.167} C_VEL
LIN {X 0,Y 128.917,Z 187.427,A -85,B 0,C 180,E1 -25240.858,E2 -25240.858} C_VEL
LIN {X 0,Y 128.984,Z 187.419,A -85,B 0,C 180,E1 -25247.939,E2 -25247.939} C_VEL
LIN {X 0,Y 130.887,Z 192.45,A -85,B 0,C 180,E1 -25248.74,E2 -25248.74} C_VEL
LIN {X 0,Y 133.655,Z 199.593,A -85,B 0,C 180,E1 -25249.826,E2 -25249.826} C_VEL
LIN {X 0,Y 140.419,Z 222.213,A -85,B 0,C 180,E1 -25252.71,E2 -25252.71} C_VEL
LIN {X 0,Y 141.777,Z 227.826,A -85,B 0,C 180,E1 -25253.335,E2 -25253.335} C_VEL
LIN {X 0,Y 143.046,Z 243.061,A -85,B 0,C 180,E1 -25254.666,E2 -25254.666} C_VEL
LIN {X 0,Y 139.48,Z 293.113,A -85,B 0,C 180,E1 -25258.167,E2 -25258.167} C_VEL
LIN {X 0,Y 137.955,Z 307.212,A -85,B 0,C 180,E1 -25259.722,E2 -25259.722} C_VEL
LIN {X 0,Y 136.088,Z 319.809,A -85,B 0,C 180,E1 -25261.693,E2 -25261.693} C_VEL
LIN {X 0,Y 133.996,Z 332.424,A -85,B 0,C 180,E1 -25264.364,E2 -25264.364} C_VEL
LIN {X 0,Y 132.031,Z 343.2,A -85,B 0,C 180,E1 -25267.302,E2 -25267.302} C_VEL
LIN {X 0,Y 130.094,Z 354.044,A -85,B 0,C 180,E1 -25271.09,E2 -25271.09} C_VEL
LIN {X 0,Y 128.59,Z 362.848,A -85,B 0,C 180,E1 -25274.956,E2 -25274.956} C_VEL
LIN {X 0,Y 127.589,Z 371.451,A -85,B 0,C 180,E1 -25279.69,E2 -25279.69} C_VEL
LIN {X 0,Y 127.128,Z 378.975,A -85,B 0,C 180,E1 -25285.008,E2 -25285.008} C_VEL
LIN {X 0,Y 127.127,Z 384.433,A -85,B 0,C 180,E1 -25290.003,E2 -25290.003} C_VEL
LIN {X 0,Y 126.879,Z 388.016,A -85,B 0,C 180,E1 -25294.409,E2 -25294.409} C_VEL
LIN {X 0,Y 127.11,Z 391.086,A -85,B 0,C 180,E1 -25299.551,E2 -25299.551} C_VEL
LIN {X 0,Y 128.781,Z 393.514,A -85,B 0,C 180,E1 -25305.838,E2 -25305.838} C_VEL
LIN {X 0,Y 131.908,Z 394.478,A -85,B 0,C 180,E1 -25311.901,E2 -25311.901} C_VEL
LIN {X 0,Y 136.838,Z 394.039,A -85,B 0,C 180,E1 -25317.534,E2 -25317.534} C_VEL
LIN {X 0,Y 143.105,Z 392.21,A -85,B 0,C 180,E1 -25322.701,E2 -25322.701} C_VEL
LIN {X 0,Y 150.44,Z 388.94,A -85,B 0,C 180,E1 -25327.398,E2 -25327.398} C_VEL
LIN {X 0,Y 153.389,Z 387.37,A -85,B 0,C 180,E1 -25328.937,E2 -25328.937} C_VEL
LIN {X 0,Y 156.319,Z 385.542,A -85,B 0,C 180,E1 -25330.715,E2 -25330.715} C_VEL
LIN {X 0,Y 160.129,Z 382.429,A -85,B 0,C 180,E1 -25333.837,E2 -25333.837} C_VEL
LIN {X 0,Y 164.318,Z 378.786,A -85,B 0,C 180,E1 -25336.716,E2 -25336.716} C_VEL
LIN {X 0,Y 167.723,Z 376.123,A -85,B 0,C 180,E1 -25338.09,E2 -25338.09} C_VEL
LIN {X 0,Y 177.179,Z 368.462,A -85,B 0,C 180,E1 -25340.671,E2 -25340.671} C_VEL
LIN {X 0,Y 185.652,Z 360.358,A -85,B 0,C 180,E1 -25342.655,E2 -25342.655} C_VEL
LIN {X 0,Y 194.43,Z 350.406,A -85,B 0,C 180,E1 -25344.422,E2 -25344.422} C_VEL
LIN {X 0,Y 201.993,Z 340.248,A -85,B 0,C 180,E1 -25345.727,E2 -25345.727} C_VEL
LIN {X 0,Y 208.987,Z 329.052,A -85,B 0,C 180,E1 -25346.777,E2 -25346.777} C_VEL
LIN {X 0,Y 215.219,Z 316.801,A -85,B 0,C 180,E1 -25347.584,E2 -25347.584} C_VEL
LIN {X 0,Y 220.203,Z 304.293,A -85,B 0,C 180,E1 -25348.224,E2 -25348.224} C_VEL
LIN {X 0,Y 220.934,Z 302.103,A -85,B 0,C 180,E1 -25348.312,E2 -25348.312} C_VEL
LIN {X 0,Y 221.521,Z 300.284,A -85,B 0,C 180,E1 -25348.525,E2 -25348.525} C_VEL
LIN {X 0,Y 221.553,Z 300.03,A -85,B 0,C 180,E1 -25349.878,E2 -25349.878} C_VEL
LIN {X 0,Y 220.945,Z 301.902,A -85,B 0,C 180,E1 -25350.165,E2 -25350.165} C_VEL
LIN {X 0,Y 215.833,Z 315.179,A -85,B 0,C 180,E1 -25350.896,E2 -25350.896} C_VEL
LIN {X 0,Y 210.088,Z 326.691,A -85,B 0,C 180,E1 -25351.802,E2 -25351.802} C_VEL
LIN {X 0,Y 202.909,Z 338.343,A -85,B 0,C 180,E1 -25353.023,E2 -25353.023} C_VEL
LIN {X 0,Y 195.438,Z 348.428,A -85,B 0,C 180,E1 -25354.436,E2 -25354.436} C_VEL
LIN {X 0,Y 187.342,Z 357.591,A -85,B 0,C 180,E1 -25356.156,E2 -25356.156} C_VEL
LIN {X 0,Y 179.234,Z 365.353,A -85,B 0,C 180,E1 -25358.13,E2 -25358.13} C_VEL
LIN {X 0,Y 170.005,Z 372.831,A -85,B 0,C 180,E1 -25360.688,E2 -25360.688} C_VEL
LIN {X 0,Y 161.134,Z 378.768,A -85,B 0,C 180,E1 -25363.655,E2 -25363.655} C_VEL
LIN {X 0,Y 153.217,Z 383.081,A -85,B 0,C 180,E1 -25366.742,E2 -25366.742} C_VEL
LIN {X 0,Y 148.294,Z 385.374,A -85,B 0,C 180,E1 -25369.073,E2 -25369.073} C_VEL
LIN {X 0,Y 141.714,Z 387.783,A -85,B 0,C 180,E1 -25372.699,E2 -25372.699} C_VEL
LIN {X 0,Y 133.585,Z 389.566,A -85,B 0,C 180,E1 -25378.464,E2 -25378.464} C_VEL
LIN {X 0,Y 127.012,Z 389.498,A -85,B 0,C 180,E1 -25385.1,E2 -25385.1} C_VEL
LIN {X 0,Y 123.771,Z 388.385,A -85,B 0,C 180,E1 -25389.809,E2 -25389.809} C_VEL
LIN {X 0,Y 121.964,Z 387.047,A -85,B 0,C 180,E1 -25393.327,E2 -25393.327} C_VEL
LIN {X 0,Y 119.772,Z 383.274,A -85,B 0,C 180,E1 -25400.133,E2 -25400.133} C_VEL
LIN {X 0,Y 119.13,Z 378.654,A -85,B 0,C 180,E1 -25406.082,E2 -25406.082} C_VEL
LIN {X 0,Y 119.44,Z 372.567,A -85,B 0,C 180,E1 -25411.978,E2 -25411.978} C_VEL
LIN {X 0,Y 120.11,Z 366.082,A -85,B 0,C 180,E1 -25416.854,E2 -25416.854} C_VEL
LIN {X 0,Y 121.29,Z 357.335,A -85,B 0,C 180,E1 -25422.078,E2 -25422.078} C_VEL
LIN {X 0,Y 122.828,Z 348.22,A -85,B 0,C 180,E1 -25426.387,E2 -25426.387} C_VEL
LIN {X 0,Y 124.66,Z 338.17,A -85,B 0,C 180,E1 -25430.189,E2 -25430.189} C_VEL
LIN {X 0,Y 126.761,Z 326.815,A -85,B 0,C 180,E1 -25433.6,E2 -25433.6} C_VEL
LIN {X 0,Y 129.002,Z 314.192,A -85,B 0,C 180,E1 -25436.491,E2 -25436.491} C_VEL
LIN {X 0,Y 130.947,Z 301.173,A -85,B 0,C 180,E1 -25438.732,E2 -25438.732} C_VEL
LIN {X 0,Y 132.429,Z 286.992,A -85,B 0,C 180,E1 -25440.443,E2 -25440.443} C_VEL
LIN {X 0,Y 134.62,Z 258.984,A -85,B 0,C 180,E1 -25442.564,E2 -25442.564} C_VEL
LIN {X 0,Y 136.896,Z 228.658,A -85,B 0,C 180,E1 -25444.701,E2 -25444.701} C_VEL
LIN {X 0,Y 133.185,Z 216.904,A -85,B 0,C 180,E1 -25446.225,E2 -25446.225} C_VEL
LIN {X 0,Y 125.129,Z 196.161,A -85,B 0,C 180,E1 -25449.385,E2 -25449.385} C_VEL
LIN {X 0,Y 122.103,Z 188.68,A -85,B 0,C 180,E1 -25450.67,E2 -25450.67} C_VEL
LIN {X 0,Y 122.048,Z 188.283,A -85,B 0,C 180,E1 -25450.879,E2 -25450.879} C_VEL
LIN {X 0,Y 122.291,Z 188.253,A -85,B 0,C 180,E1 -25457.689,E2 -25457.689} C_VEL
LIN {X 0,Y 122.399,Z 188.239,A -85,B 0,C 180,E1 -25460.078,E2 -25460.078} C_VEL
LIN {X 0,Y 122.564,Z 188.217,A -85,B 0,C 180,E1 -25466.71,E2 -25466.71} C_VEL
LIN {X 0,Y 123.024,Z 188.154,A -85,B 0,C 180,E1 -25469.997,E2 -25469.997} C_VEL
LIN {X 0,Y 122.407,Z 188.234,A -85,B 0,C 180,E1 -25476.591,E2 -25476.591} C_VEL
LIN {X 0,Y 122.391,Z 188.236,A -85,B 0,C 180,E1 -25479.917,E2 -25479.917} C_VEL
LIN {X 0,Y 122.187,Z 188.266,A -85,B 0,C 180,E1 -25483.298,E2 -25483.298} C_VEL
LIN {X 0,Y 121.986,Z 188.289,A -85,B 0,C 180,E1 -25490.22,E2 -25490.22} C_VEL
LIN {X 0,Y 121.911,Z 188.295,A -85,B 0,C 180,E1 -25493.797,E2 -25493.797} C_VEL
LIN {X 0,Y 121.914,Z 188.298,A -85,B 0,C 180,E1 -25500.148,E2 -25500.148} C_VEL
LIN {X 0,Y 121.878,Z 188.302,A -85,B 0,C 180,E1 -25506.165,E2 -25506.165} C_VEL
LIN {X 0,Y 121.86,Z 188.298,A -85,B 0,C 180,E1 -25511.43,E2 -25511.43} C_VEL
LIN {X 0,Y 121.859,Z 188.303,A -85,B 0,C 180,E1 -25518.564,E2 -25518.564} C_VEL
LIN {X 0,Y 121.903,Z 188.301,A -85,B 0,C 180,E1 -25524.792,E2 -25524.792} C_VEL
LIN {X 0,Y 121.921,Z 188.293,A -85,B 0,C 180,E1 -25529.837,E2 -25529.837} C_VEL
LIN {X 0,Y 121.98,Z 188.284,A -85,B 0,C 180,E1 -25537.191,E2 -25537.191} C_VEL
LIN {X 0,Y 122.053,Z 188.279,A -85,B 0,C 180,E1 -25543.266,E2 -25543.266} C_VEL
LIN {X 0,Y 122.281,Z 188.251,A -85,B 0,C 180,E1 -25547.69,E2 -25547.69} C_VEL
LIN {X 0,Y 122.389,Z 188.241,A -85,B 0,C 180,E1 -25550.079,E2 -25550.079} C_VEL
LIN {X 0,Y 122.554,Z 188.218,A -85,B 0,C 180,E1 -25556.712,E2 -25556.712} C_VEL
LIN {X 0,Y 123.014,Z 188.16,A -85,B 0,C 180,E1 -25559.999,E2 -25559.999} C_VEL
LIN {X 0,Y 122.398,Z 188.238,A -85,B 0,C 180,E1 -25566.594,E2 -25566.594} C_VEL
LIN {X 0,Y 122.383,Z 188.234,A -85,B 0,C 180,E1 -25569.92,E2 -25569.92} C_VEL
LIN {X 0,Y 122.179,Z 188.264,A -85,B 0,C 180,E1 -25573.302,E2 -25573.302} C_VEL
LIN {X 0,Y 121.978,Z 188.287,A -85,B 0,C 180,E1 -25580.224,E2 -25580.224} C_VEL
LIN {X 0,Y 121.904,Z 188.3,A -85,B 0,C 180,E1 -25583.8,E2 -25583.8} C_VEL
LIN {X 0,Y 121.909,Z 188.298,A -85,B 0,C 180,E1 -25590.153,E2 -25590.153} C_VEL
LIN {X 0,Y 121.874,Z 188.295,A -85,B 0,C 180,E1 -25596.17,E2 -25596.17} C_VEL
LIN {X 0,Y 121.857,Z 188.304,A -85,B 0,C 180,E1 -25601.435,E2 -25601.435} C_VEL
LIN {X 0,Y 121.885,Z 188.35,A -85,B 0,C 180,E1 -25606.654,E2 -25606.654} C_VEL
LIN {X 0,Y 122.897,Z 191.164,A -85,B 0,C 180,E1 -25607.122,E2 -25607.122} C_VEL
LIN {X 0,Y 127.157,Z 201.509,A -85,B 0,C 180,E1 -25608.863,E2 -25608.863} C_VEL
LIN {X 0,Y 134.081,Z 224.924,A -85,B 0,C 180,E1 -25611.987,E2 -25611.987} C_VEL
LIN {X 0,Y 135.116,Z 229.122,A -85,B 0,C 180,E1 -25612.488,E2 -25612.488} C_VEL
LIN {X 0,Y 136.256,Z 243.398,A -85,B 0,C 180,E1 -25613.809,E2 -25613.809} C_VEL
LIN {X 0,Y 132.602,Z 292.872,A -85,B 0,C 180,E1 -25617.436,E2 -25617.436} C_VEL
LIN {X 0,Y 131.032,Z 306.971,A -85,B 0,C 180,E1 -25619.066,E2 -25619.066} C_VEL
LIN {X 0,Y 129.129,Z 319.47,A -85,B 0,C 180,E1 -25621.119,E2 -25621.119} C_VEL
LIN {X 0,Y 127.111,Z 331.325,A -85,B 0,C 180,E1 -25623.751,E2 -25623.751} C_VEL
LIN {X 0,Y 125.099,Z 342.199,A -85,B 0,C 180,E1 -25626.846,E2 -25626.846} C_VEL
LIN {X 0,Y 123.073,Z 353.139,A -85,B 0,C 180,E1 -25630.834,E2 -25630.834} C_VEL
LIN {X 0,Y 121.544,Z 362.029,A -85,B 0,C 180,E1 -25634.921,E2 -25634.921} C_VEL
LIN {X 0,Y 120.556,Z 370.773,A -85,B 0,C 180,E1 -25639.931,E2 -25639.931} C_VEL
LIN {X 0,Y 120.129,Z 377.096,A -85,B 0,C 180,E1 -25644.488,E2 -25644.488} C_VEL
LIN {X 0,Y 120.122,Z 381.454,A -85,B 0,C 180,E1 -25648.327,E2 -25648.327} C_VEL
LIN {X 0,Y 120.112,Z 384.635,A -85,B 0,C 180,E1 -25651.679,E2 -25651.679} C_VEL
LIN {X 0,Y 119.869,Z 388.278,A -85,B 0,C 180,E1 -25656.737,E2 -25656.737} C_VEL
LIN {X 0,Y 120.893,Z 391.726,A -85,B 0,C 180,E1 -25663.449,E2 -25663.449} C_VEL
LIN {X 0,Y 123.389,Z 393.669,A -85,B 0,C 180,E1 -25669.986,E2 -25669.986} C_VEL
LIN {X 0,Y 127.777,Z 394.25,A -85,B 0,C 180,E1 -25676.108,E2 -25676.108} C_VEL
LIN {X 0,Y 133.746,Z 393.427,A -85,B 0,C 180,E1 -25681.703,E2 -25681.703} C_VEL
LIN {X 0,Y 140.917,Z 391.202,A -85,B 0,C 180,E1 -25686.764,E2 -25686.764} C_VEL
LIN {X 0,Y 147.986,Z 388.14,A -85,B 0,C 180,E1 -25690.654,E2 -25690.654} C_VEL
LIN {X 0,Y 156.228,Z 383.738,A -85,B 0,C 180,E1 -25694.212,E2 -25694.212} C_VEL
LIN {X 0,Y 163.767,Z 378.957,A -85,B 0,C 180,E1 -25696.851,E2 -25696.851} C_VEL
LIN {X 0,Y 167.723,Z 376.123,A -85,B 0,C 180,E1 -25698.09,E2 -25698.09} C_VEL
LIN {X 0,Y 171.244,Z 373.324,A -85,B 0,C 180,E1 -25699.391,E2 -25699.391} C_VEL
LIN {X 0,Y 176.142,Z 368.777,A -85,B 0,C 180,E1 -25701.813,E2 -25701.813} C_VEL
LIN {X 0,Y 181.095,Z 363.708,A -85,B 0,C 180,E1 -25704.011,E2 -25704.011} C_VEL
LIN {X 0,Y 184.586,Z 360.103,A -85,B 0,C 180,E1 -25704.965,E2 -25704.965} C_VEL
LIN {X 0,Y 193.618,Z 350.293,A -85,B 0,C 180,E1 -25706.604,E2 -25706.604} C_VEL
LIN {X 0,Y 201.415,Z 340.227,A -85,B 0,C 180,E1 -25707.799,E2 -25707.799} C_VEL
LIN {X 0,Y 208.59,Z 329.017,A -85,B 0,C 180,E1 -25708.758,E2 -25708.758} C_VEL
LIN {X 0,Y 212.66,Z 321.508,A -85,B 0,C 180,E1 -25709.235,E2 -25709.235} C_VEL
LIN {X 0,Y 212.127,Z 322.496,A -85,B 0,C 180,E1 -25709.478,E2 -25709.478} C_VEL
LIN {X 0,Y 205.241,Z 334.372,A -85,B 0,C 180,E1 -25710.513,E2 -25710.513} C_VEL
LIN {X 0,Y 197.797,Z 344.78,A -85,B 0,C 180,E1 -25711.706,E2 -25711.706} C_VEL
LIN {X 0,Y 189.915,Z 353.979,A -85,B 0,C 180,E1 -25713.159,E2 -25713.159} C_VEL
LIN {X 0,Y 180.594,Z 363.183,A -85,B 0,C 180,E1 -25715.098,E2 -25715.098} C_VEL
LIN {X 0,Y 170.353,Z 371.463,A -85,B 0,C 180,E1 -25717.567,E2 -25717.567} C_VEL
LIN {X 0,Y 162.658,Z 376.657,A -85,B 0,C 180,E1 -25719.779,E2 -25719.779} C_VEL
LIN {X 0,Y 154.884,Z 381.133,A -85,B 0,C 180,E1 -25722.35,E2 -25722.35} C_VEL
LIN {X 0,Y 145.603,Z 385.406,A -85,B 0,C 180,E1 -25726.035,E2 -25726.035} C_VEL
LIN {X 0,Y 140.606,Z 387.237,A -85,B 0,C 180,E1 -25728.468,E2 -25728.468} C_VEL
LIN {X 0,Y 134.982,Z 388.794,A -85,B 0,C 180,E1 -25731.611,E2 -25731.611} C_VEL
LIN {X 0,Y 127.525,Z 389.974,A -85,B 0,C 180,E1 -25736.841,E2 -25736.841} C_VEL
LIN {X 0,Y 124.001,Z 389.994,A -85,B 0,C 180,E1 -25740.001,E2 -25740.001} C_VEL
LIN {X 0,Y 119.867,Z 389.352,A -85,B 0,C 180,E1 -25744.598,E2 -25744.598} C_VEL
LIN {X 0,Y 115.14,Z 386.663,A -85,B 0,C 180,E1 -25752.4,E2 -25752.4} C_VEL
LIN {X 0,Y 113.129,Z 383.591,A -85,B 0,C 180,E1 -25758.097,E2 -25758.097} C_VEL
LIN {X 0,Y 112.229,Z 379.325,A -85,B 0,C 180,E1 -25764.02,E2 -25764.02} C_VEL
LIN {X 0,Y 112.271,Z 373.682,A -85,B 0,C 180,E1 -25770.053,E2 -25770.053} C_VEL
LIN {X 0,Y 112.912,Z 366.471,A -85,B 0,C 180,E1 -25775.981,E2 -25775.981} C_VEL
LIN {X 0,Y 114.046,Z 358.093,A -85,B 0,C 180,E1 -25781.403,E2 -25781.403} C_VEL
LIN {X 0,Y 115.587,Z 348.626,A -85,B 0,C 180,E1 -25786.224,E2 -25786.224} C_VEL
LIN {X 0,Y 117.45,Z 338.809,A -85,B 0,C 180,E1 -25790.188,E2 -25790.188} C_VEL
LIN {X 0,Y 119.72,Z 326.679,A -85,B 0,C 180,E1 -25794.05,E2 -25794.05} C_VEL
LIN {X 0,Y 121.99,Z 314.267,A -85,B 0,C 180,E1 -25797.033,E2 -25797.033} C_VEL
LIN {X 0,Y 123.9,Z 301.811,A -85,B 0,C 180,E1 -25799.299,E2 -25799.299} C_VEL
LIN {X 0,Y 125.456,Z 287.815,A -85,B 0,C 180,E1 -25801.099,E2 -25801.099} C_VEL
LIN {X 0,Y 127.4,Z 264.121,A -85,B 0,C 180,E1 -25803.031,E2 -25803.031} C_VEL
LIN {X 0,Y 130.125,Z 229.98,A -85,B 0,C 180,E1 -25805.579,E2 -25805.579} C_VEL
LIN {X 0,Y 126.716,Z 219.285,A -85,B 0,C 180,E1 -25807.042,E2 -25807.042} C_VEL
LIN {X 0,Y 118.878,Z 198.867,A -85,B 0,C 180,E1 -25810.372,E2 -25810.372} C_VEL
LIN {X 0,Y 115.053,Z 189.566,A -85,B 0,C 180,E1 -25812.087,E2 -25812.087} C_VEL
LIN {X 0,Y 115.005,Z 189.161,A -85,B 0,C 180,E1 -25812.206,E2 -25812.206} C_VEL
LIN {X 0,Y 115.312,Z 189.122,A -85,B 0,C 180,E1 -25819.462,E2 -25819.462} C_VEL
LIN {X 0,Y 115.491,Z 189.098,A -85,B 0,C 180,E1 -25826.508,E2 -25826.508} C_VEL
LIN {X 0,Y 115.976,Z 189.032,A -85,B 0,C 180,E1 -25829.997,E2 -25829.997} C_VEL
LIN {X 0,Y 115.349,Z 189.114,A -85,B 0,C 180,E1 -25836.996,E2 -25836.996} C_VEL
LIN {X 0,Y 115.205,Z 189.134,A -85,B 0,C 180,E1 -25842.554,E2 -25842.554} C_VEL
LIN {X 0,Y 114.963,Z 189.16,A -85,B 0,C 180,E1 -25847.795,E2 -25847.795} C_VEL
LIN {X 0,Y 114.892,Z 189.17,A -85,B 0,C 180,E1 -25853.426,E2 -25853.426} C_VEL
LIN {X 0,Y 114.845,Z 189.178,A -85,B 0,C 180,E1 -25861.046,E2 -25861.046} C_VEL
LIN {X 0,Y 114.772,Z 189.188,A -85,B 0,C 180,E1 -25867.755,E2 -25867.755} C_VEL
LIN {X 0,Y 114.775,Z 189.181,A -85,B 0,C 180,E1 -25872.708,E2 -25872.708} C_VEL
LIN {X 0,Y 114.782,Z 189.186,A -85,B 0,C 180,E1 -25877.659,E2 -25877.659} C_VEL
LIN {X 0,Y 114.779,Z 189.186,A -85,B 0,C 180,E1 -25882.744,E2 -25882.744} C_VEL
LIN {X 0,Y 114.85,Z 189.173,A -85,B 0,C 180,E1 -25888.942,E2 -25888.942} C_VEL
LIN {X 0,Y 114.901,Z 189.166,A -85,B 0,C 180,E1 -25896.554,E2 -25896.554} C_VEL
LIN {X 0,Y 114.958,Z 189.166,A -85,B 0,C 180,E1 -25902.2,E2 -25902.2} C_VEL
LIN {X 0,Y 115.302,Z 189.122,A -85,B 0,C 180,E1 -25909.463,E2 -25909.463} C_VEL
LIN {X 0,Y 115.481,Z 189.1,A -85,B 0,C 180,E1 -25916.51,E2 -25916.51} C_VEL
LIN {X 0,Y 115.966,Z 189.038,A -85,B 0,C 180,E1 -25919.999,E2 -25919.999} C_VEL
LIN {X 0,Y 115.34,Z 189.117,A -85,B 0,C 180,E1 -25926.999,E2 -25926.999} C_VEL
LIN {X 0,Y 115.197,Z 189.133,A -85,B 0,C 180,E1 -25932.556,E2 -25932.556} C_VEL
LIN {X 0,Y 114.956,Z 189.16,A -85,B 0,C 180,E1 -25937.799,E2 -25937.799} C_VEL
LIN {X 0,Y 114.886,Z 189.175,A -85,B 0,C 180,E1 -25943.43,E2 -25943.43} C_VEL
LIN {X 0,Y 114.841,Z 189.18,A -85,B 0,C 180,E1 -25951.05,E2 -25951.05} C_VEL
LIN {X 0,Y 114.768,Z 189.185,A -85,B 0,C 180,E1 -25957.76,E2 -25957.76} C_VEL
LIN {X 0,Y 114.783,Z 189.189,A -85,B 0,C 180,E1 -25964.804,E2 -25964.804} C_VEL
LIN {X 0,Y 114.823,Z 189.377,A -85,B 0,C 180,E1 -25965.24,E2 -25965.24} C_VEL
LIN {X 0,Y 116.705,Z 194.101,A -85,B 0,C 180,E1 -25966.119,E2 -25966.119} C_VEL
LIN {X 0,Y 120.906,Z 204.179,A -85,B 0,C 180,E1 -25967.945,E2 -25967.945} C_VEL
LIN {X 0,Y 127.641,Z 227.354,A -85,B 0,C 180,E1 -25971.21,E2 -25971.21} C_VEL
LIN {X 0,Y 128.558,Z 231.645,A -85,B 0,C 180,E1 -25971.722,E2 -25971.722} C_VEL
LIN {X 0,Y 129.409,Z 244.881,A -85,B 0,C 180,E1 -25972.98,E2 -25972.98} C_VEL
LIN {X 0,Y 125.673,Z 293.237,A -85,B 0,C 180,E1 -25976.756,E2 -25976.756} C_VEL
LIN {X 0,Y 123.985,Z 307.507,A -85,B 0,C 180,E1 -25978.529,E2 -25978.529} C_VEL
LIN {X 0,Y 122.054,Z 319.767,A -85,B 0,C 180,E1 -25980.7,E2 -25980.7} C_VEL
LIN {X 0,Y 119.959,Z 331.502,A -85,B 0,C 180,E1 -25983.47,E2 -25983.47} C_VEL
LIN {X 0,Y 117.929,Z 342.316,A -85,B 0,C 180,E1 -25986.749,E2 -25986.749} C_VEL
LIN {X 0,Y 116.062,Z 352.207,A -85,B 0,C 180,E1 -25990.549,E2 -25990.549} C_VEL
LIN {X 0,Y 114.498,Z 361.211,A -85,B 0,C 180,E1 -25994.882,E2 -25994.882} C_VEL
LIN {X 0,Y 113.523,Z 370.065,A -85,B 0,C 180,E1 -26000.201,E2 -26000.201} C_VEL
LIN {X 0,Y 113.122,Z 377.059,A -85,B 0,C 180,E1 -26005.581,E2 -26005.581} C_VEL
LIN {X 0,Y 113.158,Z 381.668,A -85,B 0,C 180,E1 -26010.003,E2 -26010.003} C_VEL
LIN {X 0,Y 113.012,Z 384.673,A -85,B 0,C 180,E1 -26013.568,E2 -26013.568} C_VEL
LIN {X 0,Y 113.247,Z 389.213,A -85,B 0,C 180,E1 -26020.733,E2 -26020.733} C_VEL
LIN {X 0,Y 115.209,Z 392.195,A -85,B 0,C 180,E1 -26027.762,E2 -26027.762} C_VEL
LIN {X 0,Y 118.857,Z 393.727,A -85,B 0,C 180,E1 -26034.454,E2 -26034.454} C_VEL
LIN {X 0,Y 124.398,Z 393.896,A -85,B 0,C 180,E1 -26040.565,E2 -26040.565} C_VEL
LIN {X 0,Y 131.396,Z 392.713,A -85,B 0,C 180,E1 -26046.044,E2 -26046.044} C_VEL
LIN {X 0,Y 139.476,Z 390.151,A -85,B 0,C 180,E1 -26050.927,E2 -26050.927} C_VEL
LIN {X 0,Y 148.807,Z 386.086,A -85,B 0,C 180,E1 -26055.111,E2 -26055.111} C_VEL
LIN {X 0,Y 156.432,Z 381.973,A -85,B 0,C 180,E1 -26057.845,E2 -26057.845} C_VEL
LIN {X 0,Y 167.233,Z 374.936,A -85,B 0,C 180,E1 -26061.032,E2 -26061.032} C_VEL
LIN {X 0,Y 177.184,Z 367.02,A -85,B 0,C 180,E1 -26063.441,E2 -26063.441} C_VEL
LIN {X 0,Y 184.586,Z 360.103,A -85,B 0,C 180,E1 -26064.965,E2 -26064.965} C_VEL
LIN {X 0,Y 186.89,Z 357.677,A -85,B 0,C 180,E1 -26065.64,E2 -26065.64} C_VEL
LIN {X 0,Y 193.029,Z 350.496,A -85,B 0,C 180,E1 -26068.558,E2 -26068.558} C_VEL
LIN {X 0,Y 195.247,Z 347.774,A -85,B 0,C 180,E1 -26069.102,E2 -26069.102} C_VEL
LIN {X 0,Y 196.273,Z 346.504,A -85,B 0,C 180,E1 -26069.25,E2 -26069.25} C_VEL
LIN {X 0,Y 195.771,Z 347.085,A -85,B 0,C 180,E1 -26069.829,E2 -26069.829} C_VEL
LIN {X 0,Y 187.241,Z 356.453,A -85,B 0,C 180,E1 -26071.292,E2 -26071.292} C_VEL
LIN {X 0,Y 178.168,Z 364.705,A -85,B 0,C 180,E1 -26073.024,E2 -26073.024} C_VEL
LIN {X 0,Y 168.031,Z 372.399,A -85,B 0,C 180,E1 -26075.276,E2 -26075.276} C_VEL
LIN {X 0,Y 159.82,Z 377.611,A -85,B 0,C 180,E1 -26077.443,E2 -26077.443} C_VEL
LIN {X 0,Y 149.251,Z 383.045,A -85,B 0,C 180,E1 -26080.755,E2 -26080.755} C_VEL
LIN {X 0,Y 143.396,Z 385.456,A -85,B 0,C 180,E1 -26082.899,E2 -26082.899} C_VEL
LIN {X 0,Y 138.001,Z 387.347,A -85,B 0,C 180,E1 -26085.249,E2 -26085.249} C_VEL
LIN {X 0,Y 132.902,Z 388.732,A -85,B 0,C 180,E1 -26087.789,E2 -26087.789} C_VEL
LIN {X 0,Y 128.091,Z 389.666,A -85,B 0,C 180,E1 -26090.527,E2 -26090.527} C_VEL
LIN {X 0,Y 123.705,Z 390.182,A -85,B 0,C 180,E1 -26093.476,E2 -26093.476} C_VEL
LIN {X 0,Y 119.683,Z 390.272,A -85,B 0,C 180,E1 -26096.673,E2 -26096.673} C_VEL
LIN {X 0,Y 116.162,Z 389.902,A -85,B 0,C 180,E1 -26100.001,E2 -26100.001} C_VEL
LIN {X 0,Y 112.73,Z 389.006,A -85,B 0,C 180,E1 -26104.017,E2 -26104.017} C_VEL
LIN {X 0,Y 110.492,Z 387.943,A -85,B 0,C 180,E1 -26107.309,E2 -26107.309} C_VEL
LIN {X 0,Y 107.925,Z 385.724,A -85,B 0,C 180,E1 -26112.356,E2 -26112.356} C_VEL
LIN {X 0,Y 105.758,Z 381.575,A -85,B 0,C 180,E1 -26119.408,E2 -26119.408} C_VEL
LIN {X 0,Y 105.088,Z 376.653,A -85,B 0,C 180,E1 -26125.768,E2 -26125.768} C_VEL
LIN {X 0,Y 105.421,Z 370.132,A -85,B 0,C 180,E1 -26132.232,E2 -26132.232} C_VEL
LIN {X 0,Y 106.232,Z 362.691,A -85,B 0,C 180,E1 -26138.008,E2 -26138.008} C_VEL
LIN {X 0,Y 107.508,Z 353.997,A -85,B 0,C 180,E1 -26143.386,E2 -26143.386} C_VEL
LIN {X 0,Y 109.389,Z 343.879,A -85,B 0,C 180,E1 -26148.323,E2 -26148.323} C_VEL
LIN {X 0,Y 111.556,Z 332.29,A -85,B 0,C 180,E1 -26152.748,E2 -26152.748} C_VEL
LIN {X 0,Y 113.917,Z 320.167,A -85,B 0,C 180,E1 -26156.269,E2 -26156.269} C_VEL
LIN {X 0,Y 116.197,Z 307.152,A -85,B 0,C 180,E1 -26159.107,E2 -26159.107} C_VEL
LIN {X 0,Y 117.895,Z 294.339,A -85,B 0,C 180,E1 -26161.134,E2 -26161.134} C_VEL
LIN {X 0,Y 119.307,Z 280.251,A -85,B 0,C 180,E1 -26162.651,E2 -26162.651} C_VEL
LIN {X 0,Y 123.366,Z 231.554,A -85,B 0,C 180,E1 -26166.495,E2 -26166.495} C_VEL
LIN {X 0,Y 120.542,Z 222.27,A -85,B 0,C 180,E1 -26167.84,E2 -26167.84} C_VEL
LIN {X 0,Y 112.566,Z 201.382,A -85,B 0,C 180,E1 -26171.453,E2 -26171.453} C_VEL
LIN {X 0,Y 108.086,Z 190.809,A -85,B 0,C 180,E1 -26173.592,E2 -26173.592} C_VEL
LIN {X 0,Y 107.958,Z 190.039,A -85,B 0,C 180,E1 -26173.815,E2 -26173.815} C_VEL
LIN {X 0,Y 108.231,Z 190.004,A -85,B 0,C 180,E1 -26178.763,E2 -26178.763} C_VEL
LIN {X 0,Y 108.294,Z 189.995,A -85,B 0,C 180,E1 -26182.539,E2 -26182.539} C_VEL
LIN {X 0,Y 108.901,Z 189.913,A -85,B 0,C 180,E1 -26189.997,E2 -26189.997} C_VEL
LIN {X 0,Y 108.288,Z 189.99,A -85,B 0,C 180,E1 -26197.455,E2 -26197.455} C_VEL
LIN {X 0,Y 108.138,Z 190.015,A -85,B 0,C 180,E1 -26202.869,E2 -26202.869} C_VEL
LIN {X 0,Y 107.86,Z 190.047,A -85,B 0,C 180,E1 -26209.01,E2 -26209.01} C_VEL
LIN {X 0,Y 107.801,Z 190.052,A -85,B 0,C 180,E1 -26214.114,E2 -26214.114} C_VEL
LIN {X 0,Y 107.771,Z 190.057,A -85,B 0,C 180,E1 -26222.029,E2 -26222.029} C_VEL
LIN {X 0,Y 107.681,Z 190.072,A -85,B 0,C 180,E1 -26228.443,E2 -26228.443} C_VEL
LIN {X 0,Y 107.666,Z 190.073,A -85,B 0,C 180,E1 -26235.888,E2 -26235.888} C_VEL
LIN {X 0,Y 107.679,Z 190.068,A -85,B 0,C 180,E1 -26241.551,E2 -26241.551} C_VEL
LIN {X 0,Y 107.786,Z 190.052,A -85,B 0,C 180,E1 -26248.557,E2 -26248.557} C_VEL
LIN {X 0,Y 107.867,Z 190.041,A -85,B 0,C 180,E1 -26256.987,E2 -26256.987} C_VEL
LIN {X 0,Y 107.961,Z 190.03,A -85,B 0,C 180,E1 -26264.906,E2 -26264.906} C_VEL
LIN {X 0,Y 108.219,Z 190.005,A -85,B 0,C 180,E1 -26268.764,E2 -26268.764} C_VEL
LIN {X 0,Y 108.284,Z 189.992,A -85,B 0,C 180,E1 -26272.541,E2 -26272.541} C_VEL
LIN {X 0,Y 108.892,Z 189.919,A -85,B 0,C 180,E1 -26279.999,E2 -26279.999} C_VEL
LIN {X 0,Y 108.279,Z 189.998,A -85,B 0,C 180,E1 -26287.458,E2 -26287.458} C_VEL
LIN {X 0,Y 108.13,Z 190.013,A -85,B 0,C 180,E1 -26292.871,E2 -26292.871} C_VEL
LIN {X 0,Y 107.852,Z 190.043,A -85,B 0,C 180,E1 -26299.014,E2 -26299.014} C_VEL
LIN {X 0,Y 107.795,Z 190.057,A -85,B 0,C 180,E1 -26304.117,E2 -26304.117} C_VEL
LIN {X 0,Y 107.766,Z 190.061,A -85,B 0,C 180,E1 -26312.034,E2 -26312.034} C_VEL
LIN {X 0,Y 107.677,Z 190.07,A -85,B 0,C 180,E1 -26318.448,E2 -26318.448} C_VEL
LIN {X 0,Y 107.72,Z 190.105,A -85,B 0,C 180,E1 -26323.64,E2 -26323.64} C_VEL
LIN {X 0,Y 109.606,Z 194.921,A -85,B 0,C 180,E1 -26324.607,E2 -26324.607} C_VEL
LIN {X 0,Y 114.589,Z 206.649,A -85,B 0,C 180,E1 -26326.905,E2 -26326.905} C_VEL
LIN {X 0,Y 121.096,Z 229.315,A -85,B 0,C 180,E1 -26330.318,E2 -26330.318} C_VEL
LIN {X 0,Y 121.919,Z 233.139,A -85,B 0,C 180,E1 -26330.809,E2 -26330.809} C_VEL
LIN {X 0,Y 122.598,Z 245.862,A -85,B 0,C 180,E1 -26332.076,E2 -26332.076} C_VEL
LIN {X 0,Y 118.857,Z 292.456,A -85,B 0,C 180,E1 -26335.894,E2 -26335.894} C_VEL
LIN {X 0,Y 117.242,Z 305.886,A -85,B 0,C 180,E1 -26337.609,E2 -26337.609} C_VEL
LIN {X 0,Y 115.296,Z 318.174,A -85,B 0,C 180,E1 -26339.812,E2 -26339.812} C_VEL
LIN {X 0,Y 113.45,Z 328.698,A -85,B 0,C 180,E1 -26342.319,E2 -26342.319} C_VEL
LIN {X 0,Y 111.005,Z 341.18,A -85,B 0,C 180,E1 -26346.199,E2 -26346.199} C_VEL
LIN {X 0,Y 109.059,Z 351.225,A -85,B 0,C 180,E1 -26350.229,E2 -26350.229} C_VEL
LIN {X 0,Y 107.477,Z 360.303,A -85,B 0,C 180,E1 -26354.841,E2 -26354.841} C_VEL
LIN {X 0,Y 106.501,Z 369.196,A -85,B 0,C 180,E1 -26360.508,E2 -26360.508} C_VEL
LIN {X 0,Y 106.139,Z 376.277,A -85,B 0,C 180,E1 -26366.207,E2 -26366.207} C_VEL
LIN {X 0,Y 106.192,Z 381.82,A -85,B 0,C 180,E1 -26371.9,E2 -26371.9} C_VEL
LIN {X 0,Y 105.978,Z 385.956,A -85,B 0,C 180,E1 -26377.625,E2 -26377.625} C_VEL
LIN {X 0,Y 107.209,Z 389.959,A -85,B 0,C 180,E1 -26385.205,E2 -26385.205} C_VEL
LIN {X 0,Y 110.15,Z 392.479,A -85,B 0,C 180,E1 -26392.512,E2 -26392.512} C_VEL
LIN {X 0,Y 115.209,Z 393.656,A -85,B 0,C 180,E1 -26399.214,E2 -26399.214} C_VEL
LIN {X 0,Y 121.902,Z 393.483,A -85,B 0,C 180,E1 -26405.21,E2 -26405.21} C_VEL
LIN {X 0,Y 129.833,Z 391.926,A -85,B 0,C 180,E1 -26410.513,E2 -26410.513} C_VEL
LIN {X 0,Y 134.211,Z 390.649,A -85,B 0,C 180,E1 -26412.906,E2 -26412.906} C_VEL
LIN {X 0,Y 143.936,Z 386.99,A -85,B 0,C 180,E1 -26417.092,E2 -26417.092} C_VEL
LIN {X 0,Y 151.832,Z 383.218,A -85,B 0,C 180,E1 -26419.799,E2 -26419.799} C_VEL
LIN {X 0,Y 160.127,Z 378.488,A -85,B 0,C 180,E1 -26422.191,E2 -26422.191} C_VEL
LIN {X 0,Y 169.068,Z 372.427,A -85,B 0,C 180,E1 -26424.361,E2 -26424.361} C_VEL
LIN {X 0,Y 178.838,Z 364.637,A -85,B 0,C 180,E1 -26426.394,E2 -26426.394} C_VEL
LIN {X 0,Y 188.427,Z 355.45,A -85,B 0,C 180,E1 -26428.056,E2 -26428.056} C_VEL
LIN {X 0,Y 195.247,Z 347.774,A -85,B 0,C 180,E1 -26429.102,E2 -26429.102} C_VEL
LIN {X 0,Y 194.274,Z 348.886,A -85,B 0,C 180,E1 -26429.311,E2 -26429.311} C_VEL
LIN {X 0,Y 189.163,Z 354.454,A -85,B 0,C 180,E1 -26429.323,E2 -26429.323} C_VEL
LIN {X 0,Y 180.994,Z 362.268,A -85,B 0,C 180,E1 -26428.849,E2 -26428.849} C_VEL
LIN {X 0,Y 174.711,Z 367.525,A -85,B 0,C 180,E1 -26428.151,E2 -26428.151} C_VEL
LIN {X 0,Y 172.638,Z 369.1,A -85,B 0,C 180,E1 -26427.806,E2 -26427.806} C_VEL
LIN {X 0,Y 161.825,Z 376.574,A -85,B 0,C 180,E1 -26425.608,E2 -26425.608} C_VEL
LIN {X 0,Y 150.214,Z 383.038,A -85,B 0,C 180,E1 -26422.694,E2 -26422.694} C_VEL
LIN {X 0,Y 139.247,Z 387.839,A -85,B 0,C 180,E1 -26419.21,E2 -26419.21} C_VEL
LIN {X 0,Y 129.125,Z 391.097,A -85,B 0,C 180,E1 -26415.041,E2 -26415.041} C_VEL
LIN {X 0,Y 120.212,Z 392.945,A -85,B 0,C 180,E1 -26410.027,E2 -26410.027} C_VEL
LIN {X 0,Y 112.392,Z 393.472,A -85,B 0,C 180,E1 -26404.252,E2 -26404.252} C_VEL
LIN {X 0,Y 106.113,Z 392.677,A -85,B 0,C 180,E1 -26397.625,E2 -26397.625} C_VEL
LIN {X 0,Y 101.814,Z 390.55,A -85,B 0,C 180,E1 -26390.194,E2 -26390.194} C_VEL
LIN {X 0,Y 99.507,Z 386.969,A -85,B 0,C 180,E1 -26382.236,E2 -26382.236} C_VEL
LIN {X 0,Y 99.124,Z 381.841,A -85,B 0,C 180,E1 -26374.069,E2 -26374.069} C_VEL
LIN {X 0,Y 99.242,Z 378.494,A -85,B 0,C 180,E1 -26370.003,E2 -26370.003} C_VEL
LIN {X 0,Y 99.202,Z 372.87,A -85,B 0,C 180,E1 -26364.544,E2 -26364.544} C_VEL
LIN {X 0,Y 99.726,Z 365.534,A -85,B 0,C 180,E1 -26358.829,E2 -26358.829} C_VEL
LIN {X 0,Y 101.088,Z 355.821,A -85,B 0,C 180,E1 -26352.818,E2 -26352.818} C_VEL
LIN {X 0,Y 102.914,Z 345.722,A -85,B 0,C 180,E1 -26347.943,E2 -26347.943} C_VEL
LIN {X 0,Y 105.182,Z 334.543,A -85,B 0,C 180,E1 -26343.73,E2 -26343.73} C_VEL
LIN {X 0,Y 107.302,Z 323.813,A -85,B 0,C 180,E1 -26340.582,E2 -26340.582} C_VEL
LIN {X 0,Y 109.498,Z 311.036,A -85,B 0,C 180,E1 -26337.76,E2 -26337.76} C_VEL
LIN {X 0,Y 111.474,Z 297.144,A -85,B 0,C 180,E1 -26335.571,E2 -26335.571} C_VEL
LIN {X 0,Y 113.026,Z 280.709,A -85,B 0,C 180,E1 -26333.934,E2 -26333.934} C_VEL
LIN {X 0,Y 115.925,Z 243.996,A -85,B 0,C 180,E1 -26330.816,E2 -26330.816} C_VEL
LIN {X 0,Y 115.018,Z 232.871,A -85,B 0,C 180,E1 -26329.564,E2 -26329.564} C_VEL
LIN {X 0,Y 109.057,Z 211.759,A -85,B 0,C 180,E1 -26326.258,E2 -26326.258} C_VEL
LIN {X 0,Y 107.058,Z 205.966,A -85,B 0,C 180,E1 -26325.195,E2 -26325.195} C_VEL
LIN {X 0,Y 100.823,Z 191.666,A -85,B 0,C 180,E1 -26321.99,E2 -26321.99} C_VEL
LIN {X 0,Y 100.675,Z 190.942,A -85,B 0,C 180,E1 -26321.734,E2 -26321.734} C_VEL
LIN {X 0,Y 100.678,Z 190.943,A -85,B 0,C 180,E1 -26313.111,E2 -26313.111} C_VEL
LIN {X 0,Y 100.718,Z 190.938,A -85,B 0,C 180,E1 -26304.75,E2 -26304.75} C_VEL
LIN {X 0,Y 100.766,Z 190.93,A -85,B 0,C 180,E1 -26300.409,E2 -26300.409} C_VEL
LIN {X 0,Y 101.108,Z 190.886,A -85,B 0,C 180,E1 -26292.035,E2 -26292.035} C_VEL
LIN {X 0,Y 101.214,Z 190.876,A -85,B 0,C 180,E1 -26287.982,E2 -26287.982} C_VEL
LIN {X 0,Y 101.819,Z 190.799,A -85,B 0,C 180,E1 -26279.999,E2 -26279.999} C_VEL
LIN {X 0,Y 101.221,Z 190.873,A -85,B 0,C 180,E1 -26272.017,E2 -26272.017} C_VEL
LIN {X 0,Y 101.044,Z 190.894,A -85,B 0,C 180,E1 -26266.827,E2 -26266.827} C_VEL
LIN {X 0,Y 100.772,Z 190.93,A -85,B 0,C 180,E1 -26259.591,E2 -26259.591} C_VEL
LIN {X 0,Y 100.729,Z 190.935,A -85,B 0,C 180,E1 -26255.089,E2 -26255.089} C_VEL
LIN {X 0,Y 100.683,Z 190.94,A -85,B 0,C 180,E1 -26246.885,E2 -26246.885} C_VEL
LIN {X 0,Y 100.63,Z 190.943,A -85,B 0,C 180,E1 -26240.19,E2 -26240.19} C_VEL
LIN {X 0,Y 100.637,Z 190.947,A -85,B 0,C 180,E1 -26234.29,E2 -26234.29} C_VEL
LIN {X 0,Y 100.619,Z 190.951,A -85,B 0,C 180,E1 -26228.944,E2 -26228.944} C_VEL
LIN {X 0,Y 100.682,Z 190.937,A -85,B 0,C 180,E1 -26223.106,E2 -26223.106} C_VEL
LIN {X 0,Y 100.724,Z 190.932,A -85,B 0,C 180,E1 -26214.746,E2 -26214.746} C_VEL
LIN {X 0,Y 100.773,Z 190.932,A -85,B 0,C 180,E1 -26210.404,E2 -26210.404} C_VEL
LIN {X 0,Y 101.116,Z 190.89,A -85,B 0,C 180,E1 -26202.032,E2 -26202.032} C_VEL
LIN {X 0,Y 101.222,Z 190.869,A -85,B 0,C 180,E1 -26197.979,E2 -26197.979} C_VEL
LIN {X 0,Y 101.829,Z 190.794,A -85,B 0,C 180,E1 -26189.997,E2 -26189.997} C_VEL
LIN {X 0,Y 101.231,Z 190.877,A -85,B 0,C 180,E1 -26182.015,E2 -26182.015} C_VEL
LIN {X 0,Y 101.074,Z 190.896,A -85,B 0,C 180,E1 -26176.777,E2 -26176.777} C_VEL
LIN {X 0,Y 100.963,Z 190.91,A -85,B 0,C 180,E1 -26175.498,E2 -26175.498} C_VEL
LIN {X 0,Y 102.786,Z 195.824,A -85,B 0,C 180,E1 -26174.391,E2 -26174.391} C_VEL
LIN {X 0,Y 108.559,Z 209.607,A -85,B 0,C 180,E1 -26171.472,E2 -26171.472} C_VEL
LIN {X 0,Y 115.721,Z 229.268,A -85,B 0,C 180,E1 -26168.065,E2 -26168.065} C_VEL
LIN {X 0,Y 116.563,Z 232.05,A -85,B 0,C 180,E1 -26167.637,E2 -26167.637} C_VEL
LIN {X 0,Y 111.97,Z 285.445,A -85,B 0,C 180,E1 -26163.084,E2 -26163.084} C_VEL
LIN {X 0,Y 110.405,Z 299.208,A -85,B 0,C 180,E1 -26161.235,E2 -26161.235} C_VEL
LIN {X 0,Y 108.327,Z 312.37,A -85,B 0,C 180,E1 -26158.73,E2 -26158.73} C_VEL
LIN {X 0,Y 105.808,Z 325.481,A -85,B 0,C 180,E1 -26155.285,E2 -26155.285} C_VEL
LIN {X 0,Y 103.548,Z 336.97,A -85,B 0,C 180,E1 -26151.311,E2 -26151.311} C_VEL
LIN {X 0,Y 101.43,Z 347.867,A -85,B 0,C 180,E1 -26146.423,E2 -26146.423} C_VEL
LIN {X 0,Y 100.029,Z 355.994,A -85,B 0,C 180,E1 -26141.873,E2 -26141.873} C_VEL
LIN {X 0,Y 98.994,Z 363.389,A -85,B 0,C 180,E1 -26136.824,E2 -26136.824} C_VEL
LIN {X 0,Y 98.307,Z 370.353,A -85,B 0,C 180,E1 -26130.914,E2 -26130.914} C_VEL
LIN {X 0,Y 98.125,Z 375.535,A -85,B 0,C 180,E1 -26125.452,E2 -26125.452} C_VEL
LIN {X 0,Y 98.851,Z 380.749,A -85,B 0,C 180,E1 -26118.66,E2 -26118.66} C_VEL
LIN {X 0,Y 100.805,Z 384.726,A -85,B 0,C 180,E1 -26112.074,E2 -26112.074} C_VEL
LIN {X 0,Y 102.754,Z 386.759,A -85,B 0,C 180,E1 -26107.863,E2 -26107.863} C_VEL
LIN {X 0,Y 105.611,Z 388.467,A -85,B 0,C 180,E1 -26103.392,E2 -26103.392} C_VEL
LIN {X 0,Y 111.885,Z 390.218,A -85,B 0,C 180,E1 -26096.399,E2 -26096.399} C_VEL
LIN {X 0,Y 115.886,Z 390.537,A -85,B 0,C 180,E1 -26093.034,E2 -26093.034} C_VEL
LIN {X 0,Y 121.7,Z 390.296,A -85,B 0,C 180,E1 -26089.044,E2 -26089.044} C_VEL
LIN {X 0,Y 131.796,Z 388.551,A -85,B 0,C 180,E1 -26083.717,E2 -26083.717} C_VEL
LIN {X 0,Y 141.717,Z 385.546,A -85,B 0,C 180,E1 -26079.688,E2 -26079.688} C_VEL
LIN {X 0,Y 151.14,Z 381.64,A -85,B 0,C 180,E1 -26076.717,E2 -26076.717} C_VEL
LIN {X 0,Y 160.924,Z 376.51,A -85,B 0,C 180,E1 -26074.105,E2 -26074.105} C_VEL
LIN {X 0,Y 169.487,Z 371.085,A -85,B 0,C 180,E1 -26072.193,E2 -26072.193} C_VEL
LIN {X 0,Y 178.64,Z 364.176,A -85,B 0,C 180,E1 -26070.411,E2 -26070.411} C_VEL
LIN {X 0,Y 181.851,Z 361.416,A -85,B 0,C 180,E1 -26069.841,E2 -26069.841} C_VEL
LIN {X 0,Y 180.182,Z 362.934,A -85,B 0,C 180,E1 -26069.108,E2 -26069.108} C_VEL
